KUKA KRL program: MyProgram_273().src

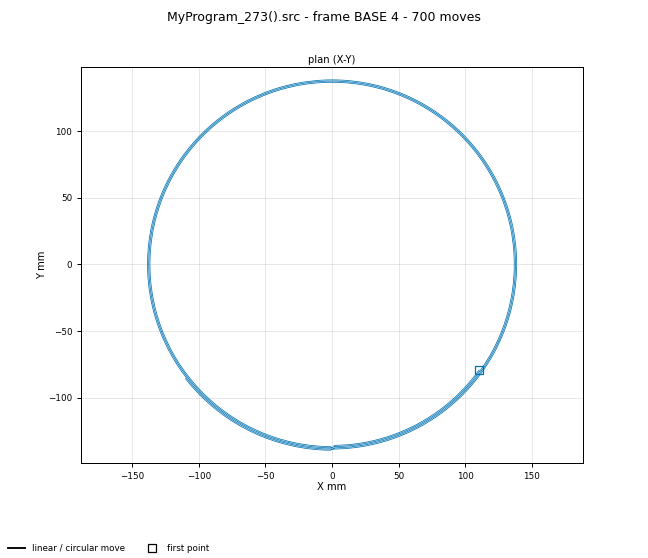
[picture p0: tool path of MyProgram_273().src in frame BASE 4, 700 of 700 moves have a stored position in this frame; points joined in program order, loops and branches not executed]
&ACCESS RVP
&REL 1
&PARAM TEMPLATE = C:\KRC\Roboter\Template\vorgabe
&PARAM EDITMASK = *
DEF MyProgram_273()
; ---- Setting reference (Base) ----
$BASE = BASE_DATA[4]

; --------------------------
; ---- Setting tool (TCP) ----
$TOOL = TOOL_DATA[3]
; --------------------------

$VEL.CP = VEL_APROX_PRINT
Startdeposition()
$VEL.CP = VEL_PRINT
LIN {X 110.2888,Y -79.2997,Z 171,A -34.2093,B 9.0943,C 0.3127,E1 9.2291,E2 485.5867} C_DIS
LIN {X 107.672,Y -82.8179,Z 171,A -36.0735,B 9.0942,C 0.3174,E1 9.226,E2 487.4547} C_DIS
LIN {X 104.9459,Y -86.2463,Z 171,A -37.9185,B 9.094,C 0.3216,E1 9.2227,E2 489.3013} C_DIS
LIN {X 101.9868,Y -89.7259,Z 171,A -39.7835,B 9.094,C 0.3246,E1 9.2193,E2 491.1605} C_DIS
LIN {X 99.052,Y -92.9557,Z 171,A -41.6097,B 9.0938,C 0.3284,E1 9.2159,E2 492.9868} C_DIS
LIN {X 95.9836,Y -96.1207,Z 171,A -43.5121,B 9.0936,C 0.3333,E1 9.2121,E2 494.8965} C_DIS
LIN {X 92.5375,Y -99.4422,Z 171,A -45.3676,B 9.0936,C 0.3339,E1 9.2084,E2 496.7335} C_DIS
LIN {X 89.5014,Y -102.1836,Z 171,A -47.1413,B 9.0934,C 0.3385,E1 9.2047,E2 498.5149} C_DIS
LIN {X 85.9377,Y -105.1981,Z 171,A -48.9197,B 9.0934,C 0.3381,E1 9.2009,E2 500.2713} C_DIS
LIN {X 82.826,Y -107.6658,Z 171,A -50.7547,B 9.0932,C 0.3448,E1 9.1968,E2 502.128} C_DIS
LIN {X 79.3157,Y -110.2774,Z 171,A -52.4701,B 9.0932,C 0.3453,E1 9.193,E2 503.8288} C_DIS
LIN {X 75.9025,Y -112.6536,Z 171,A -54.2813,B 9.093,C 0.3496,E1 9.1888,E2 505.6489} C_DIS
LIN {X 72.1992,Y -115.0623,Z 171,A -56.1436,B 9.0929,C 0.3526,E1 9.1844,E2 507.5127} C_DIS
LIN {X 69.2091,Y -116.8853,Z 171,A -57.4543,B 9.0929,C 0.3514,E1 9.1813,E2 508.8038} C_DIS
LIN {X 63.7335,Y -119.9577,Z 171,A -60.1603,B 9.0927,C 0.3567,E1 9.1747,E2 511.5193} C_DIS
LIN {X 60.3824,Y -121.6777,Z 171,A -61.7388,B 9.0927,C 0.3587,E1 9.1708,E2 513.0978} C_DIS
LIN {X 56.7536,Y -123.4119,Z 171,A -63.423,B 9.0926,C 0.3607,E1 9.1665,E2 514.7819} C_DIS
LIN {X 52.7255,Y -125.1862,Z 171,A -65.2144,B 9.0926,C 0.3617,E1 9.1619,E2 516.5666} C_DIS
LIN {X 50.0864,Y -126.2669,Z 171,A -66.5978,B 9.0923,C 0.3669,E1 9.1583,E2 517.9737} C_DIS
LIN {X 46.1854,Y -127.7433,Z 171,A -68.2377,B 9.0923,C 0.3664,E1 9.154,E2 519.6} C_DIS
LIN {X 42.2838,Y -129.0888,Z 171,A -70.0071,B 9.0923,C 0.3688,E1 9.1493,E2 521.3743} C_DIS
LIN {X 38.5569,Y -130.2496,Z 171,A -71.5883,B 9.0923,C 0.369,E1 9.1451,E2 522.9485} C_DIS
LIN {X 34.9122,Y -131.273,Z 171,A -73.1237,B 9.0923,C 0.3691,E1 9.141,E2 524.4773} C_DIS
LIN {X 31.5826,Y -132.1138,Z 171,A -74.6101,B 9.0922,C 0.3711,E1 9.137,E2 525.9694} C_DIS
LIN {X 27.5255,Y -133.0189,Z 171,A -76.3575,B 9.0922,C 0.3723,E1 9.1322,E2 527.7172} C_DIS
LIN {X 23.8817,Y -133.7204,Z 171,A -77.8272,B 9.0922,C 0.3713,E1 9.1282,E2 529.176} C_DIS
LIN {X 20.5645,Y -134.2708,Z 171,A -79.3166,B 9.0921,C 0.3736,E1 9.124,E2 530.6751} C_DIS
LIN {X 16.385,Y -134.8448,Z 171,A -81.052,B 9.0921,C 0.3736,E1 9.1193,E2 532.406} C_DIS
LIN {X 13.6701,Y -135.1485,Z 171,A -82.6176,B 9.0917,C 0.3824,E1 9.1148,E2 534.0241} C_DIS
LIN {X 9.9582,Y -135.4709,Z 171,A -83.7269,B 9.0921,C 0.3737,E1 9.1118,E2 535.0764} C_DIS
LIN {X 2.0076,Y -135.8219,Z 171,A -87.0574,B 9.0921,C 0.374,E1 9.1026,E2 538.4055} C_DIS
LIN {X 2.0076,Y -135.8219,Z 171,A -87.0574,B 9.0921,C 0.374,E1 9.1026,E2 538.4055} C_DIS
Enddeposition()
LIN {X 0.9917,Y -136.7415,Z 171,A -87.0539,B 9.0534,C 0.3716,E1 9.0639,E2 538.3927} C_DIS
Startdeposition()
$VEL.CP = VEL_PRINT
LIN {X 3.873,Y -136.6919,Z 171,A -85.7411,B 9.0534,C 0.3693,E1 9.0676,E2 537.066} C_DIS
LIN {X 6.7914,Y -136.578,Z 171,A -84.4615,B 9.0535,C 0.3678,E1 9.0711,E2 535.7785} C_DIS
LIN {X 10.0316,Y -136.3783,Z 171,A -83.129,B 9.0535,C 0.368,E1 9.0749,E2 534.4488} C_DIS
LIN {X 13.3491,Y -136.0938,Z 171,A -81.6253,B 9.0537,C 0.3652,E1 9.0791,E2 532.9305} C_DIS
LIN {X 16.9828,Y -135.6903,Z 171,A -80.2042,B 9.0536,C 0.3668,E1 9.083,E2 531.5227} C_DIS
LIN {X 20.1333,Y -135.2587,Z 171,A -78.8736,B 9.0536,C 0.3661,E1 9.0867,E2 530.1915} C_DIS
LIN {X 23.2971,Y -134.7498,Z 171,A -77.533,B 9.0536,C 0.3653,E1 9.0904,E2 528.8504} C_DIS
LIN {X 26.4717,Y -134.1623,Z 171,A -76.04,B 9.0538,C 0.3615,E1 9.0945,E2 527.3386} C_DIS
LIN {X 29.8951,Y -133.4399,Z 171,A -74.6788,B 9.0538,C 0.3626,E1 9.0982,E2 525.9898} C_DIS
LIN {X 33.2548,Y -132.6419,Z 171,A -73.4363,B 9.0536,C 0.3657,E1 9.1015,E2 524.7724} C_DIS
LIN {X 36.0325,Y -131.9164,Z 171,A -71.9412,B 9.0539,C 0.3585,E1 9.1056,E2 523.2391} C_DIS
LIN {X 39.6821,Y -130.8626,Z 171,A -70.6296,B 9.0537,C 0.3629,E1 9.109,E2 521.9621} C_DIS
LIN {X 42.4081,Y -130.007,Z 171,A -69.3026,B 9.0539,C 0.359,E1 9.1126,E2 520.6177} C_DIS
LIN {X 45.5874,Y -128.9266,Z 171,A -67.9022,B 9.0539,C 0.3576,E1 9.1163,E2 519.217} C_DIS
LIN {X 48.7566,Y -127.7617,Z 171,A -66.4946,B 9.054,C 0.3562,E1 9.12,E2 517.8093} C_DIS
LIN {X 52.3424,Y -126.3328,Z 171,A -64.8676,B 9.054,C 0.354,E1 9.1242,E2 516.1798} C_DIS
LIN {X 55.0524,Y -125.1778,Z 171,A -63.6596,B 9.0541,C 0.353,E1 9.1273,E2 514.9741} C_DIS
LIN {X 58.1724,Y -123.7588,Z 171,A -62.2327,B 9.0541,C 0.3513,E1 9.1309,E2 513.5473} C_DIS
LIN {X 61.2693,Y -122.2552,Z 171,A -60.6628,B 9.0544,C 0.3466,E1 9.1349,E2 511.9597} C_DIS
LIN {X 65.1029,Y -120.2576,Z 171,A -58.8989,B 9.0544,C 0.3449,E1 9.1392,E2 510.2003} C_DIS
LIN {X 68.8887,Y -118.1297,Z 171,A -57.0932,B 9.0545,C 0.3424,E1 9.1436,E2 508.3949} C_DIS
LIN {X 72.6202,Y -115.8731,Z 171,A -55.281,B 9.0546,C 0.3398,E1 9.1479,E2 506.583} C_DIS
LIN {X 76.291,Y -113.4899,Z 171,A -53.4633,B 9.0547,C 0.337,E1 9.1521,E2 504.7656} C_DIS
LIN {X 79.8947,Y -110.9825,Z 171,A -51.6558,B 9.0548,C 0.3344,E1 9.1562,E2 502.9605} C_DIS
LIN {X 83.4251,Y -108.3537,Z 171,A -49.8295,B 9.0549,C 0.3314,E1 9.1603,E2 501.1348} C_DIS
LIN {X 86.8762,Y -105.6068,Z 171,A -48.0005,B 9.0551,C 0.3283,E1 9.1643,E2 499.3065} C_DIS
LIN {X 90.2421,Y -102.7455,Z 171,A -46.1693,B 9.0551,C 0.3251,E1 9.1681,E2 497.476} C_DIS
LIN {X 93.5172,Y -99.7738,Z 171,A -44.3222,B 9.0553,C 0.3214,E1 9.1719,E2 495.6278} C_DIS
LIN {X 96.6961,Y -96.6961,Z 171,A -42.5051,B 9.0554,C 0.3183,E1 9.1755,E2 493.8135} C_DIS
LIN {X 99.7738,Y -93.5172,Z 171,A -40.6587,B 9.0555,C 0.3144,E1 9.1791,E2 491.9663} C_DIS
LIN {X 102.7455,Y -90.2421,Z 171,A -38.8292,B 9.0557,C 0.3108,E1 9.1825,E2 490.1379} C_DIS
LIN {X 105.6068,Y -86.8762,Z 171,A -37.0024,B 9.0557,C 0.3071,E1 9.1858,E2 488.3123} C_DIS
LIN {X 108.3537,Y -83.4251,Z 171,A -35.1793,B 9.0559,C 0.3033,E1 9.1889,E2 486.4905} C_DIS
LIN {X 110.9825,Y -79.8947,Z 171,A -33.3758,B 9.056,C 0.2998,E1 9.1919,E2 484.6903} C_DIS
LIN {X 113.4899,Y -76.291,Z 171,A -31.5625,B 9.0562,C 0.2959,E1 9.1947,E2 482.8785} C_DIS
LIN {X 115.8731,Y -72.6202,Z 171,A -29.7557,B 9.0562,C 0.2919,E1 9.1974,E2 481.0731} C_DIS
LIN {X 118.1297,Y -68.8887,Z 171,A -27.956,B 9.0564,C 0.2879,E1 9.2,E2 479.2751} C_DIS
LIN {X 120.2576,Y -65.1029,Z 171,A -26.1847,B 9.0565,C 0.2843,E1 9.2024,E2 477.508} C_DIS
LIN {X 122.2552,Y -61.2693,Z 171,A -24.4684,B 9.0566,C 0.2817,E1 9.2045,E2 475.8019} C_DIS
LIN {X 123.7588,Y -58.1724,Z 171,A -23.0371,B 9.0567,C 0.2781,E1 9.2063,E2 474.3705} C_DIS
LIN {X 125.1778,Y -55.0524,Z 171,A -21.6354,B 9.0568,C 0.275,E1 9.2079,E2 472.9717} C_DIS
LIN {X 126.6723,Y -51.5156,Z 171,A -20.0199,B 9.057,C 0.2704,E1 9.2096,E2 471.3536} C_DIS
LIN {X 127.8921,Y -48.4084,Z 171,A -18.8127,B 9.057,C 0.271,E1 9.2108,E2 470.1693} C_DIS
LIN {X 128.9266,Y -45.5874,Z 171,A -17.4388,B 9.0571,C 0.2649,E1 9.2121,E2 468.7795} C_DIS
LIN {X 130.1445,Y -41.9777,Z 171,A -15.9362,B 9.0571,C 0.2626,E1 9.2134,E2 467.287} C_DIS
LIN {X 131.0034,Y -39.2221,Z 171,A -14.6802,B 9.0573,C 0.2581,E1 9.2144,E2 466.0239} C_DIS
LIN {X 131.9164,Y -36.0325,Z 171,A -13.3137,B 9.0574,C 0.2547,E1 9.2155,E2 464.659} C_DIS
LIN {X 132.7466,Y -32.8423,Z 171,A -11.9562,B 9.0574,C 0.2514,E1 9.2164,E2 463.3031} C_DIS
LIN {X 133.4949,Y -29.6544,Z 171,A -10.4872,B 9.0577,C 0.2452,E1 9.2173,E2 461.8204} C_DIS
LIN {X 134.1623,Y -26.4717,Z 171,A -9.2693,B 9.0577,C 0.2446,E1 9.218,E2 460.6194} C_DIS
LIN {X 134.7498,Y -23.2971,Z 171,A -7.9402,B 9.0577,C 0.2413,E1 9.2186,E2 459.292} C_DIS
LIN {X 135.2587,Y -20.1333,Z 171,A -6.6214,B 9.0579,C 0.238,E1 9.2192,E2 457.9749} C_DIS
LIN {X 135.7338,Y -16.6182,Z 171,A -5.2956,B 9.0579,C 0.2374,E1 9.2197,E2 456.6678} C_DIS
LIN {X 136.0459,Y -13.8481,Z 171,A -4.0144,B 9.058,C 0.2314,E1 9.22,E2 455.3712} C_DIS
LIN {X 136.3272,Y -10.7317,Z 171,A -2.6901,B 9.0581,C 0.2273,E1 9.2204,E2 454.044} C_DIS
LIN {X 136.5356,Y -7.6359,Z 171,A -1.4498,B 9.0581,C 0.2249,E1 9.2206,E2 452.81} C_DIS
LIN {X 136.6728,Y -4.5627,Z 171,A -0.0223,B 9.0584,C 0.2179,E1 9.2207,E2 451.3637} C_DIS
LIN {X 136.7472,Y -0.5669,Z 171,A 1.3911,B 9.0584,C 0.2191,E1 9.2207,E2 449.9817} C_DIS
LIN {X 136.7291,Y 2.201,Z 171,A 2.6312,B 9.0584,C 0.2138,E1 9.2207,E2 448.7303} C_DIS
LIN {X 136.6458,Y 5.2551,Z 171,A 3.866,B 9.0585,C 0.2112,E1 9.2207,E2 447.5} C_DIS
LIN {X 136.4833,Y 8.4834,Z 171,A 5.2015,B 9.0585,C 0.2077,E1 9.2204,E2 446.1657} C_DIS
LIN {X 136.239,Y 11.7759,Z 171,A 6.6115,B 9.0587,C 0.2031,E1 9.2201,E2 444.7511} C_DIS
LIN {X 135.8775,Y 15.4133,Z 171,A 8.0744,B 9.0587,C 0.2002,E1 9.2196,E2 443.2956} C_DIS
LIN {X 135.4537,Y 18.7684,Z 171,A 9.3927,B 9.0588,C 0.1984,E1 9.2192,E2 441.9885} C_DIS
LIN {X 135.014,Y 21.7137,Z 171,A 10.832,B 9.059,C 0.1905,E1 9.2185,E2 440.524} C_DIS
LIN {X 134.3733,Y 25.3678,Z 171,A 12.2748,B 9.059,C 0.1886,E1 9.2178,E2 439.0939} C_DIS
LIN {X 133.4949,Y 29.6544,Z 171,A 14.0413,B 9.059,C 0.1849,E1 9.2168,E2 437.3344} C_DIS
LIN {X 132.6344,Y 33.2844,Z 171,A 15.5539,B 9.0591,C 0.1817,E1 9.2158,E2 435.8268} C_DIS
LIN {X 131.8569,Y 36.2452,Z 171,A 16.8542,B 9.0592,C 0.1777,E1 9.2149,E2 434.5233} C_DIS
LIN {X 131.0034,Y 39.2221,Z 171,A 18.1264,B 9.0592,C 0.1747,E1 9.2139,E2 433.2533} C_DIS
LIN {X 129.8916,Y 42.7547,Z 171,A 19.6534,B 9.0594,C 0.171,E1 9.2126,E2 431.7282} C_DIS
LIN {X 128.9266,Y 45.5874,Z 171,A 20.8926,B 9.0594,C 0.1679,E1 9.2114,E2 430.49} C_DIS
LIN {X 127.7617,Y 48.7566,Z 171,A 22.375,B 9.0595,C 0.1626,E1 9.2099,E2 428.9981} C_DIS
LIN {X 126.5122,Y 51.9128,Z 171,A 23.6906,B 9.0595,C 0.1612,E1 9.2086,E2 427.6949} C_DIS
LIN {X 124.9735,Y 55.5093,Z 171,A 25.2436,B 9.0595,C 0.1588,E1 9.2069,E2 426.1515} C_DIS
LIN {X 123.5373,Y 58.636,Z 171,A 26.5408,B 9.0595,C 0.1582,E1 9.2054,E2 424.8714} C_DIS
LIN {X 122.0945,Y 61.5849,Z 171,A 28.0933,B 9.0597,C 0.1507,E1 9.2034,E2 423.2959} C_DIS
LIN {X 120.276,Y 65.0685,Z 171,A 29.8184,B 9.0598,C 0.1448,E1 9.2011,E2 421.5601} C_DIS
LIN {X 118.0845,Y 68.9655,Z 171,A 31.6414,B 9.0598,C 0.1412,E1 9.1986,E2 419.7423} C_DIS
LIN {X 115.8731,Y 72.6202,Z 171,A 33.4486,B 9.0599,C 0.1365,E1 9.1959,E2 417.932} C_DIS
LIN {X 113.4899,Y 76.291,Z 171,A 35.2409,B 9.0599,C 0.133,E1 9.1932,E2 416.1439} C_DIS
LIN {X 110.9825,Y 79.8947,Z 171,A 37.0651,B 9.06,C 0.129,E1 9.1902,E2 414.3206} C_DIS
LIN {X 108.3537,Y 83.4251,Z 171,A 38.8844,B 9.06,C 0.1254,E1 9.1872,E2 412.5036} C_DIS
LIN {X 105.6068,Y 86.8762,Z 171,A 40.6901,B 9.0601,C 0.1222,E1 9.184,E2 410.7024} C_DIS
LIN {X 102.7455,Y 90.2421,Z 171,A 42.5256,B 9.0601,C 0.1185,E1 9.1807,E2 408.8681} C_DIS
LIN {X 99.7738,Y 93.5172,Z 171,A 44.3659,B 9.0602,C 0.1149,E1 9.1772,E2 407.0287} C_DIS
LIN {X 96.6961,Y 96.6961,Z 171,A 46.1837,B 9.0602,C 0.1119,E1 9.1736,E2 405.2147} C_DIS
LIN {X 93.5172,Y 99.7738,Z 171,A 48.0321,B 9.0603,C 0.1083,E1 9.1699,E2 403.3664} C_DIS
LIN {X 90.2421,Y 102.7455,Z 171,A 49.8651,B 9.0603,C 0.1052,E1 9.1661,E2 401.5354} C_DIS
LIN {X 86.8172,Y 105.655,Z 171,A 51.7094,B 9.0603,C 0.1026,E1 9.1621,E2 399.6955} C_DIS
LIN {X 83.4182,Y 108.3589,Z 171,A 53.527,B 9.0604,C 0.0995,E1 9.1581,E2 397.8777} C_DIS
LIN {X 79.8947,Y 110.9825,Z 171,A 55.3362,B 9.0604,C 0.097,E1 9.154,E2 396.0721} C_DIS
LIN {X 76.291,Y 113.4899,Z 171,A 57.158,B 9.0604,C 0.0944,E1 9.1499,E2 394.2522} C_DIS
LIN {X 72.6202,Y 115.8731,Z 171,A 58.9746,B 9.0604,C 0.092,E1 9.1456,E2 392.4375} C_DIS
LIN {X 68.8887,Y 118.1297,Z 171,A 60.7852,B 9.0605,C 0.0897,E1 9.1412,E2 390.6289} C_DIS
LIN {X 65.1029,Y 120.2576,Z 171,A 62.5684,B 9.0605,C 0.0879,E1 9.1369,E2 388.85} C_DIS
LIN {X 61.2693,Y 122.2552,Z 171,A 64.2972,B 9.0605,C 0.0873,E1 9.1326,E2 387.1314} C_DIS
LIN {X 57.8326,Y 123.9159,Z 171,A 65.9138,B 9.0605,C 0.085,E1 9.1285,E2 385.5126} C_DIS
LIN {X 54.7106,Y 125.3257,Z 171,A 67.1708,B 9.0605,C 0.087,E1 9.1254,E2 384.2777} C_DIS
LIN {X 51.9128,Y 126.5122,Z 171,A 68.5727,B 9.0605,C 0.083,E1 9.1217,E2 382.8601} C_DIS
LIN {X 48.7566,Y 127.7617,Z 171,A 69.9852,B 9.0605,C 0.0817,E1 9.118,E2 381.4489} C_DIS
LIN {X 45.1805,Y 129.0676,Z 171,A 71.5897,B 9.0606,C 0.08,E1 9.1138,E2 379.8434} C_DIS
LIN {X 41.8719,Y 130.1783,Z 171,A 72.9371,B 9.0606,C 0.0811,E1 9.1103,E2 378.5103} C_DIS
LIN {X 39.2221,Y 131.0034,Z 171,A 74.179,B 9.0606,C 0.0785,E1 9.1069,E2 377.2589} C_DIS
LIN {X 36.0325,Y 131.9164,Z 171,A 75.7095,B 9.0606,C 0.0746,E1 9.1028,E2 375.7114} C_DIS
LIN {X 32.348,Y 132.8657,Z 171,A 76.9585,B 9.0606,C 0.0805,E1 9.0995,E2 374.5051} C_DIS
LIN {X 29.6544,Y 133.4949,Z 171,A 78.3001,B 9.0606,C 0.0761,E1 9.0958,E2 373.1414} C_DIS
LIN {X 26.4717,Y 134.1623,Z 171,A 79.8045,B 9.0606,C 0.0725,E1 9.0916,E2 371.62} C_DIS
LIN {X 22.7916,Y 134.8341,Z 171,A 81.2261,B 9.0606,C 0.0746,E1 9.0878,E2 370.2167} C_DIS
LIN {X 18.5562,Y 135.4841,Z 171,A 83.1326,B 9.0606,C 0.0717,E1 9.0825,E2 368.2971} C_DIS
LIN {X 15.4133,Y 135.8775,Z 171,A 84.3274,B 9.0606,C 0.0739,E1 9.0792,E2 367.1191} C_DIS
LIN {X 12.2875,Y 136.1958,Z 171,A 85.8008,B 9.0606,C 0.0705,E1 9.0751,E2 365.6269} C_DIS
LIN {X 8.373,Y 136.4902,Z 171,A 87.2861,B 9.0606,C 0.0734,E1 9.071,E2 364.1617} C_DIS
LIN {X 5.2551,Y 136.6458,Z 171,A 88.5562,B 9.0606,C 0.074,E1 9.0674,E2 362.8968} C_DIS
LIN {X 2.201,Y 136.7291,Z 171,A 89.8336,B 9.0606,C 0.074,E1 9.0639,E2 361.6203} C_DIS
LIN {X -0.8306,Y 136.7443,Z 171,A 91.1056,B 9.0606,C 0.074,E1 9.0603,E2 360.3487} C_DIS
LIN {X -3.9636,Y 136.6894,Z 171,A 92.5121,B 9.0606,C 0.0723,E1 9.0564,E2 358.9313} C_DIS
LIN {X -7.6359,Y 136.5356,Z 171,A 93.9932,B 9.0606,C 0.0737,E1 9.0523,E2 357.4583} C_DIS
LIN {X -10.7317,Y 136.3272,Z 171,A 95.2974,B 9.0606,C 0.0739,E1 9.0486,E2 356.1543} C_DIS
LIN {X -13.8481,Y 136.0459,Z 171,A 96.6132,B 9.0606,C 0.0742,E1 9.045,E2 354.8386} C_DIS
LIN {X -16.9828,Y 135.6903,Z 171,A 98.0979,B 9.0606,C 0.0716,E1 9.0408,E2 353.3347} C_DIS
LIN {X -21.7137,Y 135.014,Z 171,A 99.951,B 9.0606,C 0.0753,E1 9.0357,E2 351.5011} C_DIS
LIN {X -24.8832,Y 134.4659,Z 171,A 101.3051,B 9.0606,C 0.0759,E1 9.032,E2 350.147} C_DIS
LIN {X -28.0622,Y 133.8386,Z 171,A 102.6696,B 9.0606,C 0.0766,E1 9.0283,E2 348.7826} C_DIS
LIN {X -31.5432,Y 133.0597,Z 171,A 104.1553,B 9.0606,C 0.0778,E1 9.0242,E2 347.2988} C_DIS
LIN {X -34.4373,Y 132.3418,Z 171,A 105.4285,B 9.0606,C 0.0783,E1 9.0208,E2 346.0235} C_DIS
LIN {X -37.6276,Y 131.4703,Z 171,A 106.9347,B 9.0606,C 0.0772,E1 9.0167,E2 344.5035} C_DIS
LIN {X -41.3181,Y 130.3552,Z 171,A 108.463,B 9.0606,C 0.0802,E1 9.0127,E2 342.987} C_DIS
LIN {X -43.9988,Y 129.4773,Z 171,A 109.6382,B 9.0606,C 0.0814,E1 9.0096,E2 341.8136} C_DIS
LIN {X -47.1734,Y 128.3547,Z 171,A 111.0588,B 9.0606,C 0.0827,E1 9.0058,E2 340.3929} C_DIS
LIN {X -50.3366,Y 127.1475,Z 171,A 112.4877,B 9.0606,C 0.084,E1 9.0021,E2 338.9637} C_DIS
LIN {X -53.4849,Y 125.8556,Z 171,A 114.0521,B 9.0606,C 0.0831,E1 8.998,E2 337.3835} C_DIS
LIN {X -56.8116,Y 124.388,Z 171,A 115.3785,B 9.0606,C 0.0885,E1 8.9947,E2 336.0824} C_DIS
LIN {X -59.7239,Y 123.0175,Z 171,A 116.8198,B 9.0606,C 0.0886,E1 8.9911,E2 334.6309} C_DIS
LIN {X -62.808,Y 121.4719,Z 171,A 118.4237,B 9.0606,C 0.0877,E1 8.987,E2 333.0087} C_DIS
LIN {X -66.6233,Y 119.422,Z 171,A 120.1989,B 9.0606,C 0.091,E1 8.9827,E2 331.2399} C_DIS
LIN {X -70.3881,Y 117.2424,Z 171,A 122.039,B 9.0605,C 0.0934,E1 8.9783,E2 329.3992} C_DIS
LIN {X -74.0961,Y 114.9349,Z 171,A 123.8868,B 9.0605,C 0.096,E1 8.9739,E2 327.5508} C_DIS
LIN {X -77.7408,Y 112.5017,Z 171,A 125.7571,B 9.0605,C 0.0984,E1 8.9696,E2 325.6779} C_DIS
LIN {X -81.316,Y 109.9453,Z 171,A 127.6025,B 9.0604,C 0.1015,E1 8.9654,E2 323.8338} C_DIS
LIN {X -84.8154,Y 107.2689,Z 171,A 129.4839,B 9.0604,C 0.1043,E1 8.9613,E2 321.9497} C_DIS
LIN {X -88.2727,Y 104.4421,Z 171,A 131.3628,B 9.0604,C 0.1077,E1 8.9572,E2 320.0716} C_DIS
LIN {X -91.5633,Y 101.5698,Z 171,A 133.2115,B 9.0603,C 0.1109,E1 8.9534,E2 318.2225} C_DIS
LIN {X -94.8006,Y 98.5552,Z 171,A 135.0865,B 9.0603,C 0.1143,E1 8.9496,E2 316.3466} C_DIS
LIN {X -97.9396,Y 95.4364,Z 171,A 136.9783,B 9.0602,C 0.1175,E1 8.9459,E2 314.452} C_DIS
LIN {X -100.9754,Y 92.2184,Z 171,A 138.8389,B 9.0602,C 0.1214,E1 8.9423,E2 312.5924} C_DIS
LIN {X -103.9035,Y 88.9063,Z 171,A 140.7299,B 9.0602,C 0.1248,E1 8.9389,E2 310.6985} C_DIS
LIN {X -106.7548,Y 85.4613,Z 171,A 142.613,B 9.06,C 0.1289,E1 8.9355,E2 308.8161} C_DIS
LIN {X -109.4196,Y 82.0221,Z 171,A 144.4705,B 9.06,C 0.1326,E1 8.9324,E2 306.9561} C_DIS
LIN {X -112.0002,Y 78.4616,Z 171,A 146.3403,B 9.06,C 0.1365,E1 8.9294,E2 305.0848} C_DIS
LIN {X -114.4775,Y 74.8007,Z 171,A 148.1925,B 9.0599,C 0.1411,E1 8.9265,E2 303.2346} C_DIS
LIN {X -116.791,Y 71.1345,Z 171,A 150.0578,B 9.0599,C 0.1448,E1 8.9238,E2 301.3651} C_DIS
LIN {X -118.9964,Y 67.3805,Z 171,A 151.9067,B 9.0597,C 0.149,E1 8.9212,E2 299.515} C_DIS
LIN {X -120.6909,Y 64.2953,Z 171,A 153.4263,B 9.0597,C 0.152,E1 8.9192,E2 297.9915} C_DIS
LIN {X -122.2552,Y 61.2693,Z 171,A 154.7436,B 9.0596,C 0.1576,E1 8.9175,E2 296.6892} C_DIS
LIN {X -123.7588,Y 58.1724,Z 171,A 156.2065,B 9.0596,C 0.1611,E1 8.9158,E2 295.2253} C_DIS
LIN {X -125.1778,Y 55.0524,Z 171,A 157.6631,B 9.0595,C 0.1646,E1 8.9141,E2 293.7676} C_DIS
LIN {X -126.6252,Y 51.6322,Z 171,A 159.127,B 9.0594,C 0.1703,E1 8.9125,E2 292.3167} C_DIS
LIN {X -127.7617,Y 48.7566,Z 171,A 160.556,B 9.0594,C 0.1716,E1 8.9111,E2 290.8726} C_DIS
LIN {X -128.9266,Y 45.5874,Z 171,A 161.9912,B 9.0593,C 0.1752,E1 8.9097,E2 289.4364} C_DIS
LIN {X -130.007,Y 42.4081,Z 171,A 163.5064,B 9.0593,C 0.1773,E1 8.9084,E2 287.9092} C_DIS
LIN {X -131.0034,Y 39.2221,Z 171,A 164.8381,B 9.0591,C 0.1823,E1 8.9073,E2 286.5873} C_DIS
LIN {X -131.9164,Y 36.0325,Z 171,A 166.2486,B 9.0591,C 0.1858,E1 8.9062,E2 285.1756} C_DIS
LIN {X -132.7466,Y 32.8423,Z 171,A 167.6503,B 9.059,C 0.1894,E1 8.9053,E2 283.7728} C_DIS
LIN {X -133.5384,Y 29.453,Z 171,A 169.052,B 9.0589,C 0.1945,E1 8.9044,E2 282.3795} C_DIS
LIN {X -134.1623,Y 26.4717,Z 171,A 170.4252,B 9.0589,C 0.1965,E1 8.9036,E2 280.9957} C_DIS
LIN {X -134.7498,Y 23.2971,Z 171,A 171.798,B 9.0588,C 0.2001,E1 8.903,E2 279.6217} C_DIS
LIN {X -135.2587,Y 20.1333,Z 171,A 173.2816,B 9.0588,C 0.2016,E1 8.9023,E2 278.122} C_DIS
LIN {X -135.7345,Y 16.6117,Z 171,A 174.664,B 9.0586,C 0.2077,E1 8.9018,E2 276.7542} C_DIS
LIN {X -136.0459,Y 13.8481,Z 171,A 175.854,B 9.0586,C 0.2106,E1 8.9015,E2 275.5624} C_DIS
LIN {X -136.3272,Y 10.7317,Z 171,A 177.1845,B 9.0584,C 0.2141,E1 8.9012,E2 274.2307} C_DIS
LIN {X -136.5356,Y 7.6359,Z 171,A 178.6029,B 9.0584,C 0.2159,E1 8.9009,E2 272.7989} C_DIS
LIN {X -136.6919,Y 3.873,Z 171,A -179.8678,B 9.0583,C 0.2213,E1 8.9008,E2 271.277} C_DIS
LIN {X -136.751,Y 0,Z 171,A -178.0171,B 9.0583,C 0.2223,E1 8.9008,E2 269.3996} C_DIS
LIN {X -136.6919,Y -3.873,Z 171,A -176.6214,B 9.058,C 0.2307,E1 8.9008,E2 268.0336} C_DIS
LIN {X -136.578,Y -6.7914,Z 171,A -175.3065,B 9.058,C 0.2328,E1 8.901,E2 266.7085} C_DIS
LIN {X -136.3509,Y -10.4062,Z 171,A -173.6956,B 9.058,C 0.2356,E1 8.9013,E2 265.0873} C_DIS
LIN {X -136.0459,Y -13.8481,Z 171,A -172.3268,B 9.0578,C 0.2411,E1 8.9017,E2 263.7296} C_DIS
LIN {X -135.6397,Y -17.3688,Z 171,A -170.7725,B 9.0577,C 0.2442,E1 8.9022,E2 262.168} C_DIS
LIN {X -135.1759,Y -20.6683,Z 171,A -169.3638,B 9.0576,C 0.248,E1 8.9028,E2 260.7588} C_DIS
LIN {X -134.4659,Y -24.8832,Z 171,A -167.5701,B 9.0575,C 0.253,E1 8.9037,E2 258.9664} C_DIS
LIN {X -133.7222,Y -28.6015,Z 171,A -165.993,B 9.0573,C 0.2577,E1 8.9046,E2 257.392} C_DIS
LIN {X -133.0445,Y -31.6062,Z 171,A -164.7795,B 9.0572,C 0.2626,E1 8.9053,E2 256.1892} C_DIS
LIN {X -132.3418,Y -34.4373,Z 171,A -163.396,B 9.0572,C 0.2634,E1 8.9063,E2 254.7865} C_DIS
LIN {X -131.4703,Y -37.6276,Z 171,A -161.9862,B 9.0571,C 0.2668,E1 8.9073,E2 253.3748} C_DIS
LIN {X -130.5157,Y -40.8158,Z 171,A -160.5124,B 9.057,C 0.2693,E1 8.9085,E2 251.8922} C_DIS
LIN {X -129.4773,Y -43.9988,Z 171,A -159.141,B 9.0569,C 0.2737,E1 8.9098,E2 250.5257} C_DIS
LIN {X -128.3547,Y -47.1734,Z 171,A -157.6095,B 9.0569,C 0.2754,E1 8.9112,E2 248.9801} C_DIS
LIN {X -127.1475,Y -50.3366,Z 171,A -156.1155,B 9.0567,C 0.2779,E1 8.9128,E2 247.4776} C_DIS
LIN {X -125.6229,Y -54.023,Z 171,A -154.5674,B 9.0565,C 0.2844,E1 8.9144,E2 245.946} C_DIS
LIN {X -124.4789,Y -56.6151,Z 171,A -153.3598,B 9.0565,C 0.2872,E1 8.9158,E2 244.7368} C_DIS
LIN {X -122.8306,Y -60.1029,Z 171,A -151.6968,B 9.0563,C 0.2905,E1 8.9178,E2 243.0689} C_DIS
LIN {X -121.4719,Y -62.808,Z 171,A -150.3396,B 9.0563,C 0.2923,E1 8.9196,E2 241.7014} C_DIS
LIN {X -119.422,Y -66.6233,Z 171,A -148.497,B 9.0561,C 0.2963,E1 8.922,E2 239.8563} C_DIS
LIN {X -117.2424,Y -70.3881,Z 171,A -146.6469,B 9.0561,C 0.3003,E1 8.9247,E2 238.0038} C_DIS
LIN {X -114.9349,Y -74.0961,Z 171,A -144.7904,B 9.0559,C 0.3042,E1 8.9275,E2 236.145} C_DIS
LIN {X -112.5017,Y -77.7408,Z 171,A -142.9071,B 9.0558,C 0.3077,E1 8.9304,E2 234.2566} C_DIS
LIN {X -109.9453,Y -81.316,Z 171,A -141.0616,B 9.0556,C 0.3119,E1 8.9335,E2 232.4115} C_DIS
LIN {X -107.2689,Y -84.8154,Z 171,A -139.1758,B 9.0556,C 0.3153,E1 8.9367,E2 230.5215} C_DIS
LIN {X -104.4235,Y -88.2946,Z 171,A -137.2888,B 9.0554,C 0.3193,E1 8.9401,E2 228.6348} C_DIS
LIN {X -101.5698,Y -91.5633,Z 171,A -135.4437,B 9.0553,C 0.3226,E1 8.9435,E2 226.787} C_DIS
LIN {X -98.5552,Y -94.8006,Z 171,A -133.5686,B 9.0551,C 0.326,E1 8.9471,E2 224.9099} C_DIS
LIN {X -95.4364,Y -97.9396,Z 171,A -131.6724,B 9.0551,C 0.3289,E1 8.9509,E2 223.009} C_DIS
LIN {X -92.2184,Y -100.9754,Z 171,A -129.8205,B 9.0549,C 0.3324,E1 8.9547,E2 221.1577} C_DIS
LIN {X -88.9052,Y -103.9044,Z 171,A -127.9336,B 9.0549,C 0.3352,E1 8.9587,E2 219.267} C_DIS
LIN {X -85.4906,Y -106.7315,Z 171,A -126.0491,B 9.0547,C 0.338,E1 8.9627,E2 217.3795} C_DIS
LIN {X -82.0221,Y -109.4196,Z 171,A -124.2182,B 9.0546,C 0.3412,E1 8.9668,E2 215.55} C_DIS
LIN {X -78.4616,Y -112.0002,Z 171,A -122.3448,B 9.0545,C 0.3435,E1 8.9711,E2 213.6729} C_DIS
LIN {X -74.8303,Y -114.4582,Z 171,A -120.5084,B 9.0544,C 0.3463,E1 8.9753,E2 211.8369} C_DIS
LIN {X -71.0992,Y -116.8124,Z 171,A -118.6414,B 9.0544,C 0.3486,E1 8.9798,E2 209.9678} C_DIS
LIN {X -67.3463,Y -119.0156,Z 171,A -116.8055,B 9.0542,C 0.3508,E1 8.9842,E2 208.1303} C_DIS
LIN {X -64.3398,Y -120.6676,Z 171,A -115.4538,B 9.0541,C 0.3543,E1 8.9875,E2 206.7896} C_DIS
LIN {X -61.1881,Y -122.2953,Z 171,A -113.9926,B 9.054,C 0.3565,E1 8.9912,E2 205.3316} C_DIS
LIN {X -57.7374,Y -123.9599,Z 171,A -112.4088,B 9.054,C 0.3588,E1 8.9951,E2 203.7505} C_DIS
LIN {X -55.0524,Y -125.1778,Z 171,A -111.1031,B 9.054,C 0.3588,E1 8.9985,E2 202.4357} C_DIS
LIN {X -51.9128,Y -126.5122,Z 171,A -109.6671,B 9.0539,C 0.3601,E1 9.0022,E2 200.9988} C_DIS
LIN {X -48.7566,Y -127.7617,Z 171,A -108.1652,B 9.0539,C 0.3599,E1 9.0061,E2 199.4866} C_DIS
LIN {X -45.3402,Y -129.0123,Z 171,A -106.6636,B 9.0538,C 0.3617,E1 9.0101,E2 197.9877} C_DIS
LIN {X -42.4081,Y -130.007,Z 171,A -105.4073,B 9.0538,C 0.3635,E1 9.0134,E2 196.7365} C_DIS
LIN {X -39.2221,Y -131.0034,Z 171,A -103.8629,B 9.0538,C 0.3617,E1 9.0176,E2 195.1732} C_DIS
LIN {X -35.9229,Y -131.9456,Z 171,A -102.606,B 9.0536,C 0.3661,E1 9.0209,E2 193.939} C_DIS
LIN {X -32.8423,Y -132.7466,Z 171,A -101.2275,B 9.0536,C 0.3661,E1 9.0246,E2 192.5545} C_DIS
LIN {X -29.6544,Y -133.4949,Z 171,A -99.7655,B 9.0536,C 0.365,E1 9.0287,E2 191.0807} C_DIS
LIN {X -25.9986,Y -134.2527,Z 171,A -98.2843,B 9.0536,C 0.3674,E1 9.0327,E2 189.6096} C_DIS
LIN {X -23.2971,Y -134.7498,Z 171,A -97.1361,B 9.0536,C 0.3679,E1 9.0358,E2 188.4615} C_DIS
LIN {X -19.5637,Y -135.3401,Z 171,A -95.7663,B 9.0534,C 0.3726,E1 9.0396,E2 187.1184} C_DIS
LIN {X -16.9828,Y -135.6903,Z 171,A -94.4614,B 9.0535,C 0.3686,E1 9.0432,E2 185.786} C_DIS
LIN {X -13.8481,Y -136.0459,Z 171,A -93.1406,B 9.0535,C 0.3689,E1 9.0469,E2 184.4648} C_DIS
LIN {X -10.7317,Y -136.3272,Z 171,A -91.831,B 9.0535,C 0.3691,E1 9.0506,E2 183.1548} C_DIS
LIN {X -7.6359,Y -136.5356,Z 171,A -90.5328,B 9.0535,C 0.3692,E1 9.0542,E2 181.8563} C_DIS
LIN {X -4.5627,Y -136.6728,Z 171,A -89.2468,B 9.0535,C 0.3692,E1 9.0578,E2 180.5702} C_DIS
LIN {X -1.5143,Y -136.7405,Z 171,A -87.8177,B 9.0536,C 0.3661,E1 9.0618,E2 179.121} C_DIS
LIN {X -1.5143,Y -136.7405,Z 171,A -87.8177,B 9.0536,C 0.3661,E1 9.0618,E2 179.121} C_DIS
Enddeposition()
LIN {X 0.999,Y -137.6517,Z 171,A -87.1205,B 9.0143,C 0.3793,E1 9.0247,E2 178.514} C_DIS
Startdeposition()
$VEL.CP = VEL_PRINT
LIN {X -2.0065,Y -137.6428,Z 171,A -88.768,B 9.0139,C 0.3874,E1 9.02,E2 180.2128} C_DIS
LIN {X -5.8902,Y -137.532,Z 171,A -90.468,B 9.0139,C 0.3891,E1 9.0152,E2 181.9242} C_DIS
LIN {X -10.1042,Y -137.2857,Z 171,A -92.1089,B 9.0139,C 0.3867,E1 9.0107,E2 183.5509} C_DIS
LIN {X -14.2208,Y -136.9214,Z 171,A -94.4711,B 9.0134,C 0.399,E1 9.0039,E2 185.9952} C_DIS
LIN {X -19.3526,Y -136.2898,Z 171,A -95.7056,B 9.0142,C 0.3805,E1 9.0008,E2 187.114} C_DIS
LIN {X -25.3246,Y -135.3084,Z 171,A -98.3818,B 9.0142,C 0.3827,E1 8.9934,E2 189.8112} C_DIS
LIN {X -29.2332,Y -134.5171,Z 171,A -100.2355,B 9.014,C 0.3857,E1 8.9882,E2 191.6901} C_DIS
LIN {X -35.4266,Y -133.0201,Z 171,A -102.5256,B 9.0144,C 0.3772,E1 8.9821,E2 193.9347} C_DIS
LIN {X -38.8817,Y -132.0516,Z 171,A -104.3105,B 9.0142,C 0.3818,E1 8.9772,E2 195.757} C_DIS
LIN {X -42.1299,Y -131.0515,Z 171,A -105.7438,B 9.0142,C 0.381,E1 8.9734,E2 197.193} C_DIS
LIN {X -45.8425,Y -129.8016,Z 171,A -107.5224,B 9.0142,C 0.3825,E1 8.9687,E2 198.9907} C_DIS
LIN {X -49.6466,Y -128.3924,Z 171,A -109.1583,B 9.0142,C 0.3799,E1 8.9644,E2 200.6201} C_DIS
LIN {X -53.1216,Y -126.9939,Z 171,A -110.7295,B 9.0142,C 0.3786,E1 8.9603,E2 202.1929} C_DIS
LIN {X -57.3013,Y -125.1645,Z 171,A -112.6269,B 9.0144,C 0.3766,E1 8.9555,E2 204.0901} C_DIS
LIN {X -60.7318,Y -123.5354,Z 171,A -114.1955,B 9.0144,C 0.3745,E1 8.9516,E2 205.6572} C_DIS
LIN {X -63.9609,Y -121.8947,Z 171,A -115.9377,B 9.0144,C 0.377,E1 8.9472,E2 207.4291} C_DIS
LIN {X -66.8955,Y -120.3118,Z 171,A -117.0895,B 9.0146,C 0.3708,E1 8.9444,E2 208.5511} C_DIS
LIN {X -70.4874,Y -118.243,Z 171,A -118.8986,B 9.0146,C 0.37,E1 8.94,E2 210.3707} C_DIS
LIN {X -74.4691,Y -115.777,Z 171,A -120.8289,B 9.0148,C 0.3669,E1 8.9355,E2 212.2984} C_DIS
LIN {X -78.1503,Y -113.3247,Z 171,A -122.7382,B 9.0148,C 0.3653,E1 8.931,E2 214.216} C_DIS
LIN {X -81.8747,Y -110.6643,Z 171,A -124.7453,B 9.0148,C 0.364,E1 8.9265,E2 216.2357} C_DIS
LIN {X -85.817,Y -107.6351,Z 171,A -126.7236,B 9.0151,C 0.3589,E1 8.9222,E2 218.2021} C_DIS
LIN {X -89.312,Y -104.7534,Z 171,A -128.6378,B 9.0152,C 0.356,E1 8.9181,E2 220.1195} C_DIS
LIN {X -92.753,Y -101.7195,Z 171,A -130.5296,B 9.0154,C 0.3522,E1 8.9141,E2 222.0085} C_DIS
LIN {X -95.9623,Y -98.6975,Z 171,A -132.4485,B 9.0154,C 0.3501,E1 8.9102,E2 223.9375} C_DIS
LIN {X -98.5779,Y -96.0856,Z 171,A -134.025,B 9.0155,C 0.3477,E1 8.9071,E2 225.5182} C_DIS
LIN {X -101.6495,Y -92.8301,Z 171,A -135.9417,B 9.0156,C 0.3448,E1 8.9035,E2 227.441} C_DIS
LIN {X -104.2352,Y -89.9161,Z 171,A -137.4907,B 9.0158,C 0.3402,E1 8.9007,E2 228.9803} C_DIS
LIN {X -107.0382,Y -86.5605,Z 171,A -139.3421,B 9.0159,C 0.3367,E1 8.8974,E2 230.8348} C_DIS
LIN {X -109.6717,Y -83.1991,Z 171,A -141.1727,B 9.0161,C 0.3337,E1 8.8942,E2 232.6713} C_DIS
LIN {X -112.3208,Y -79.5864,Z 171,A -143.0719,B 9.0161,C 0.33,E1 8.8911,E2 234.5739} C_DIS
LIN {X -114.9855,Y -75.6849,Z 171,A -145.0314,B 9.0164,C 0.3253,E1 8.8881,E2 236.5315} C_DIS
LIN {X -117.4922,Y -71.7324,Z 171,A -147.0075,B 9.0165,C 0.321,E1 8.8852,E2 238.5101} C_DIS
LIN {X -119.7219,Y -67.9459,Z 171,A -148.7613,B 9.0167,C 0.3153,E1 8.8827,E2 240.2534} C_DIS
LIN {X -122.1817,Y -63.4144,Z 171,A -150.9257,B 9.0169,C 0.3102,E1 8.8799,E2 242.4189} C_DIS
LIN {X -123.5581,Y -60.6859,Z 171,A -152.2181,B 9.0169,C 0.3073,E1 8.8783,E2 243.7129} C_DIS
LIN {X -124.9425,Y -57.7815,Z 171,A -153.6327,B 9.0171,C 0.3051,E1 8.8766,E2 245.1361} C_DIS
LIN {X -126.4786,Y -54.3379,Z 171,A -155.1801,B 9.0172,C 0.3006,E1 8.8748,E2 246.6797} C_DIS
LIN {X -127.756,Y -51.262,Z 171,A -156.6168,B 9.0173,C 0.2978,E1 8.8733,E2 248.1217} C_DIS
LIN {X -129.1906,Y -47.5372,Z 171,A -158.3747,B 9.0173,C 0.2949,E1 8.8716,E2 249.8906} C_DIS
LIN {X -130.6906,Y -43.2364,Z 171,A -160.2028,B 9.0176,C 0.2886,E1 8.8699,E2 251.7088} C_DIS
LIN {X -131.7682,Y -39.8336,Z 171,A -161.7374,B 9.0176,C 0.2854,E1 8.8687,E2 253.2484} C_DIS
LIN {X -132.8595,Y -36.0288,Z 171,A -163.4527,B 9.0178,C 0.2819,E1 8.8674,E2 254.9709} C_DIS
LIN {X -133.8205,Y -32.2716,Z 171,A -165.0378,B 9.018,C 0.2769,E1 8.8663,E2 256.551} C_DIS
LIN {X -134.6073,Y -28.8155,Z 171,A -166.5183,B 9.018,C 0.2729,E1 8.8654,E2 258.0309} C_DIS
LIN {X -135.3025,Y -25.3553,Z 171,A -168.1539,B 9.0181,C 0.2715,E1 8.8645,E2 259.6861} C_DIS
LIN {X -136.0197,Y -21.168,Z 171,A -169.8257,B 9.0183,C 0.2648,E1 8.8638,E2 261.3444} C_DIS
LIN {X -136.5146,Y -17.698,Z 171,A -171.3127,B 9.0184,C 0.2611,E1 8.8632,E2 262.8336} C_DIS
LIN {X -136.9376,Y -14.0705,Z 171,A -172.9281,B 9.0185,C 0.2583,E1 8.8627,E2 264.4595} C_DIS
LIN {X -137.2811,Y -10.1676,Z 171,A -174.5261,B 9.0187,C 0.2531,E1 8.8624,E2 266.052} C_DIS
LIN {X -137.499,Y -6.6028,Z 171,A -175.9964,B 9.0187,C 0.2485,E1 8.8621,E2 267.5189} C_DIS
LIN {X -137.6202,Y -3.2403,Z 171,A -177.5494,B 9.0188,C 0.2469,E1 8.862,E2 269.0896} C_DIS
LIN {X -137.6559,Y 0.7997,Z 171,A -179.1585,B 9.019,C 0.2409,E1 8.862,E2 270.6882} C_DIS
LIN {X -137.5937,Y 4.193,Z 171,A 179.3092,B 9.019,C 0.2387,E1 8.862,E2 272.2339} C_DIS
LIN {X -137.4131,Y 8.1959,Z 171,A 177.5308,B 9.0191,C 0.2357,E1 8.8624,E2 274.0244} C_DIS
LIN {X -137.0452,Y 12.9657,Z 171,A 175.5935,B 9.0193,C 0.229,E1 8.8628,E2 275.953} C_DIS
LIN {X -136.63,Y 16.7903,Z 171,A 174.0685,B 9.0194,C 0.2232,E1 8.8633,E2 277.4671} C_DIS
LIN {X -136.0794,Y 20.7818,Z 171,A 172.3113,B 9.0195,C 0.2196,E1 8.864,E2 279.2325} C_DIS
LIN {X -135.3835,Y 24.9238,Z 171,A 170.5903,B 9.0197,C 0.2142,E1 8.8648,E2 280.9485} C_DIS
LIN {X -134.6849,Y 28.4558,Z 171,A 169.1496,B 9.0197,C 0.209,E1 8.8656,E2 282.3805} C_DIS
LIN {X -133.9631,Y 31.6802,Z 171,A 167.5687,B 9.0197,C 0.2084,E1 8.8666,E2 283.9854} C_DIS
LIN {X -132.9524,Y 35.6803,Z 171,A 165.9145,B 9.0199,C 0.2025,E1 8.8678,E2 285.6301} C_DIS
LIN {X -131.9992,Y 39.0607,Z 171,A 164.4606,B 9.02,C 0.1983,E1 8.8689,E2 287.0815} C_DIS
LIN {X -131.0591,Y 42.1061,Z 171,A 163.1028,B 9.02,C 0.1951,E1 8.8701,E2 288.4418} C_DIS
LIN {X -130.0079,Y 45.2473,Z 171,A 161.718,B 9.0202,C 0.1914,E1 8.8713,E2 289.8258} C_DIS
LIN {X -128.805,Y 48.5664,Z 171,A 160.1796,B 9.0202,C 0.1885,E1 8.8728,E2 291.3712} C_DIS
LIN {X -127.5284,Y 51.8267,Z 171,A 158.698,B 9.0202,C 0.185,E1 8.8743,E2 292.8544} C_DIS
LIN {X -126.1932,Y 54.9979,Z 171,A 157.2295,B 9.0204,C 0.1817,E1 8.8759,E2 294.3259} C_DIS
LIN {X -124.8157,Y 58.0556,Z 171,A 155.8156,B 9.0204,C 0.1783,E1 8.8776,E2 295.7405} C_DIS
LIN {X -123.0239,Y 61.7659,Z 171,A 154.1258,B 9.0205,C 0.1734,E1 8.8797,E2 297.4254} C_DIS
LIN {X -121.6004,Y 64.5213,Z 171,A 151.6227,B 9.0202,C 0.1899,E1 8.8832,E2 300.0746} C_DIS
LIN {X -117.6996,Y 71.3913,Z 171,A 149.469,B 9.0207,C 0.163,E1 8.886,E2 302.0873} C_DIS
LIN {X -115.6362,Y 74.6876,Z 171,A 147.6989,B 9.0207,C 0.1615,E1 8.8887,E2 303.8743} C_DIS
LIN {X -113.1839,Y 78.3542,Z 171,A 145.8251,B 9.0208,C 0.1577,E1 8.8916,E2 305.7508} C_DIS
LIN {X -110.8938,Y 81.5625,Z 171,A 143.6582,B 9.0208,C 0.1626,E1 8.8953,E2 307.9802} C_DIS
LIN {X -107.8432,Y 85.5556,Z 171,A 142.0404,B 9.0209,C 0.1499,E1 8.898,E2 309.5382} C_DIS
LIN {X -104.977,Y 89.049,Z 171,A 140.154,B 9.021,C 0.1457,E1 8.9014,E2 311.4234} C_DIS
LIN {X -101.3036,Y 93.2065,Z 171,A 138.1221,B 9.0212,C 0.136,E1 8.9051,E2 313.419} C_DIS
LIN {X -99.2831,Y 95.3564,Z 171,A 136.6172,B 9.0212,C 0.1381,E1 8.9081,E2 314.9568} C_DIS
LIN {X -96.4658,Y 98.205,Z 171,A 134.8853,B 9.0212,C 0.1357,E1 8.9115,E2 316.6948} C_DIS
LIN {X -93.0203,Y 101.4748,Z 171,A 132.9535,B 9.0212,C 0.131,E1 8.9154,E2 318.6192} C_DIS
LIN {X -90.0859,Y 104.089,Z 171,A 131.2126,B 9.0212,C 0.1296,E1 8.9191,E2 320.3714} C_DIS
LIN {X -86.625,Y 106.9862,Z 171,A 129.3077,B 9.0212,C 0.1265,E1 8.9232,E2 322.2777} C_DIS
LIN {X -82.3162,Y 110.3355,Z 171,A 127.0415,B 9.0214,C 0.1224,E1 8.9282,E2 324.5412} C_DIS
LIN {X -78.7574,Y 112.9034,Z 171,A 125.2037,B 9.0214,C 0.1195,E1 8.9324,E2 326.3787} C_DIS
LIN {X -75.1407,Y 115.3421,Z 171,A 123.3058,B 9.0214,C 0.1179,E1 8.9368,E2 328.285} C_DIS
LIN {X -70.9436,Y 117.9703,Z 171,A 121.3181,B 9.0214,C 0.1135,E1 8.9415,E2 330.2619} C_DIS
LIN {X -66.4007,Y 120.5857,Z 171,A 119.2365,B 9.0215,C 0.1085,E1 8.9466,E2 332.3295} C_DIS
LIN {X -62.9151,Y 122.4389,Z 171,A 117.3585,B 9.0215,C 0.1104,E1 8.9513,E2 334.2347} C_DIS
LIN {X -59.0401,Y 124.3531,Z 171,A 115.6465,B 9.0215,C 0.1066,E1 8.9556,E2 335.9346} C_DIS
LIN {X -54.9511,Y 126.2134,Z 171,A 113.7423,B 9.0215,C 0.1049,E1 8.9604,E2 337.8415} C_DIS
LIN {X -51.2797,Y 127.7488,Z 171,A 112.1675,B 9.0216,C 0.1016,E1 8.9645,E2 339.4051} C_DIS
LIN {X -47.9208,Y 129.0469,Z 171,A 110.2611,B 9.0216,C 0.1074,E1 8.9696,E2 341.3599} C_DIS
LIN {X -44.2125,Y 130.3656,Z 171,A 108.8962,B 9.0216,C 0.1009,E1 8.9731,E2 342.6906} C_DIS
LIN {X -40.4908,Y 131.5671,Z 171,A 107.3753,B 9.0216,C 0.0974,E1 8.9771,E2 344.1971} C_DIS
LIN {X -37.0935,Y 132.5649,Z 171,A 105.8656,B 9.0216,C 0.0969,E1 8.9812,E2 345.7102} C_DIS
LIN {X -33.5681,Y 133.5015,Z 171,A 104.3541,B 9.0216,C 0.0956,E1 8.9852,E2 347.2199} C_DIS
LIN {X -30.2464,Y 134.2934,Z 171,A 102.927,B 9.0216,C 0.0948,E1 8.9891,E2 348.6468} C_DIS
LIN {X -27.0695,Y 134.9696,Z 171,A 101.583,B 9.0216,C 0.0938,E1 8.9928,E2 349.9889} C_DIS
LIN {X -22.9821,Y 135.7253,Z 171,A 99.5939,B 9.0216,C 0.0977,E1 8.9984,E2 352.0086} C_DIS
LIN {X -17.6253,Y 136.5242,Z 171,A 97.6262,B 9.0217,C 0.0914,E1 9.0037,E2 353.94} C_DIS
LIN {X -11.4473,Y 137.1803,Z 171,A 95.3312,B 9.0217,C 0.0851,E1 9.01,E2 356.198} C_DIS
LIN {X -4.2416,Y 137.5924,Z 171,A 92.1527,B 9.0217,C 0.0879,E1 9.0189,E2 359.3967} C_DIS
LIN {X 2.6091,Y 137.6328,Z 171,A 89.4103,B 9.0217,C 0.0857,E1 9.0265,E2 362.1246} C_DIS
LIN {X 9.6453,Y 137.3192,Z 171,A 86.1916,B 9.0217,C 0.0917,E1 9.0356,E2 365.3775} C_DIS
LIN {X 16.5112,Y 136.6633,Z 171,A 83.3062,B 9.0217,C 0.0927,E1 9.0436,E2 368.2637} C_DIS
LIN {X 22.036,Y 135.8831,Z 171,A 81.1089,B 9.0217,C 0.0912,E1 9.0496,E2 370.445} C_DIS
LIN {X 26.2061,Y 135.1399,Z 171,A 79.2785,B 9.0217,C 0.0934,E1 9.0547,E2 372.2831} C_DIS
LIN {X 29.3803,Y 134.4853,Z 171,A 77.5668,B 9.0217,C 0.1014,E1 9.0595,E2 374.0388} C_DIS
LIN {X 33.0614,Y 133.6301,Z 171,A 76.3665,B 9.0217,C 0.095,E1 9.0626,E2 375.1933} C_DIS
LIN {X 36.5141,Y 132.7269,Z 171,A 74.8133,B 9.0217,C 0.0975,E1 9.0668,E2 376.7545} C_DIS
LIN {X 40.3766,Y 131.6021,Z 171,A 73.1999,B 9.0217,C 0.0975,E1 9.0711,E2 378.3601} C_DIS
LIN {X 43.5144,Y 130.5981,Z 171,A 71.8599,B 9.0217,C 0.0981,E1 9.0747,E2 379.696} C_DIS
LIN {X 46.6407,Y 129.5145,Z 171,A 70.4142,B 9.0217,C 0.1008,E1 9.0785,E2 381.15} C_DIS
LIN {X 50.203,Y 128.1761,Z 171,A 68.871,B 9.0217,C 0.1016,E1 9.0825,E2 382.6881} C_DIS
LIN {X 53.4382,Y 126.8616,Z 171,A 67.4581,B 9.0216,C 0.1024,E1 9.0861,E2 384.0958} C_DIS
LIN {X 56.5853,Y 125.4895,Z 171,A 66.0339,B 9.0216,C 0.1039,E1 9.0898,E2 385.5195} C_DIS
LIN {X 59.7195,Y 124.0285,Z 171,A 64.6079,B 9.0216,C 0.1054,E1 9.0934,E2 386.9438} C_DIS
LIN {X 64.3245,Y 121.7038,Z 171,A 62.62,B 9.0216,C 0.1049,E1 9.0983,E2 388.9121} C_DIS
LIN {X 67.5458,Y 119.9477,Z 171,A 60.875,B 9.0215,C 0.1115,E1 9.1026,E2 390.6841} C_DIS
LIN {X 71.5379,Y 117.6109,Z 171,A 58.9618,B 9.0215,C 0.1141,E1 9.1072,E2 392.596} C_DIS
LIN {X 75.222,Y 115.2893,Z 171,A 57.1696,B 9.0215,C 0.1165,E1 9.1114,E2 394.3859} C_DIS
LIN {X 78.9661,Y 112.7581,Z 171,A 55.0922,B 9.0213,C 0.1236,E1 9.1162,E2 396.4877} C_DIS
LIN {X 81.6311,Y 110.8434,Z 171,A 54.1765,B 9.0214,C 0.1164,E1 9.1182,E2 397.3482} C_DIS
LIN {X 84.1447,Y 108.9477,Z 171,A 52.6198,B 9.0214,C 0.1239,E1 9.1217,E2 398.9356} C_DIS
LIN {X 87.7974,Y 106.0259,Z 171,A 50.7177,B 9.0213,C 0.1265,E1 9.1258,E2 400.8326} C_DIS
LIN {X 91.2004,Y 103.1133,Z 171,A 48.8967,B 9.0213,C 0.1291,E1 9.1296,E2 402.6488} C_DIS
LIN {X 94.3452,Y 100.2441,Z 171,A 46.9831,B 9.0212,C 0.1356,E1 9.1336,E2 404.5804} C_DIS
LIN {X 97.2997,Y 97.3796,Z 171,A 45.4238,B 9.0212,C 0.1357,E1 9.1366,E2 406.1214} C_DIS
LIN {X 102.0175,Y 92.4246,Z 171,A 42.8051,B 9.0212,C 0.1367,E1 9.1416,E2 408.7128} C_DIS
LIN {X 104.4084,Y 89.7149,Z 171,A 41.1574,B 9.0211,C 0.1431,E1 9.1447,E2 410.3788} C_DIS
LIN {X 107.1504,Y 86.4214,Z 171,A 39.3701,B 9.021,C 0.1471,E1 9.1478,E2 412.1674} C_DIS
LIN {X 109.9502,Y 82.8302,Z 171,A 37.5068,B 9.021,C 0.1507,E1 9.151,E2 414.0275} C_DIS
LIN {X 112.6465,Y 79.1246,Z 171,A 35.6104,B 9.0209,C 0.1549,E1 9.1541,E2 415.9236} C_DIS
LIN {X 115.1185,Y 75.483,Z 171,A 33.7905,B 9.0208,C 0.159,E1 9.1569,E2 417.7429} C_DIS
LIN {X 117.494,Y 71.7295,Z 171,A 31.9032,B 9.0207,C 0.1644,E1 9.1597,E2 419.636} C_DIS
LIN {X 119.9092,Y 67.6144,Z 171,A 30.0106,B 9.0207,C 0.1673,E1 9.1623,E2 421.5181} C_DIS
LIN {X 122.004,Y 63.7527,Z 171,A 28.3016,B 9.0207,C 0.1693,E1 9.1645,E2 423.2133} C_DIS
LIN {X 123.6385,Y 60.5229,Z 171,A 26.8125,B 9.0205,C 0.1728,E1 9.1664,E2 424.7011} C_DIS
LIN {X 125.2321,Y 57.1551,Z 171,A 25.2358,B 9.0205,C 0.1774,E1 9.1682,E2 426.2822} C_DIS
LIN {X 126.9578,Y 53.208,Z 171,A 23.421,B 9.0203,C 0.1826,E1 9.1702,E2 428.1007} C_DIS
LIN {X 128.2725,Y 49.9551,Z 171,A 22.0471,B 9.0203,C 0.1846,E1 9.1716,E2 429.4649} C_DIS
LIN {X 129.6314,Y 46.3164,Z 171,A 20.4987,B 9.0203,C 0.1874,E1 9.1731,E2 431.0059} C_DIS
LIN {X 130.9696,Y 42.3863,Z 171,A 18.7356,B 9.0201,C 0.193,E1 9.1747,E2 432.7747} C_DIS
LIN {X 132.149,Y 38.549,Z 171,A 17.1865,B 9.0201,C 0.1948,E1 9.1759,E2 434.3099} C_DIS
LIN {X 133.0382,Y 35.3586,Z 171,A 15.7791,B 9.02,C 0.1993,E1 9.177,E2 435.722} C_DIS
LIN {X 133.9186,Y 31.8649,Z 171,A 14.3132,B 9.02,C 0.2028,E1 9.1779,E2 437.1849} C_DIS
LIN {X 134.9065,Y 27.3796,Z 171,A 12.4612,B 9.0198,C 0.2068,E1 9.179,E2 439.031} C_DIS
LIN {X 135.5345,Y 24.0801,Z 171,A 11.0179,B 9.0198,C 0.2118,E1 9.1797,E2 440.4811} C_DIS
LIN {X 136.335,Y 19.0367,Z 171,A 9.0455,B 9.0196,C 0.2144,E1 9.1806,E2 442.4361} C_DIS
LIN {X 136.6979,Y 16.2209,Z 171,A 7.5237,B 9.0194,C 0.2256,E1 9.1811,E2 444.0016} C_DIS
LIN {X 137.0463,Y 12.9528,Z 171,A 6.5093,B 9.0194,C 0.2215,E1 9.1814,E2 444.9728} C_DIS
LIN {X 137.451,Y 7.5347,Z 171,A 4.0193,B 9.0192,C 0.2332,E1 9.1818,E2 447.4936} C_DIS
LIN {X 137.6475,Y 1.6751,Z 171,A 1.5474,B 9.019,C 0.241,E1 9.182,E2 449.9718} C_DIS
LIN {X 137.6481,Y -1.6863,Z 171,A 0.5515,B 9.0191,C 0.2359,E1 9.182,E2 450.9183} C_DIS
LIN {X 137.3528,Y -9.1756,Z 171,A -3.1491,B 9.0185,C 0.2582,E1 9.1814,E2 454.695} C_DIS
LIN {X 136.9692,Y -13.7464,Z 171,A -4.6395,B 9.0186,C 0.2542,E1 9.1811,E2 456.1347} C_DIS
LIN {X 136.5078,Y -17.7505,Z 171,A -6.6331,B 9.0183,C 0.2663,E1 9.1803,E2 458.1696} C_DIS
LIN {X 135.859,Y -22.1808,Z 171,A -8.2981,B 9.0183,C 0.2671,E1 9.1796,E2 459.8115} C_DIS
LIN {X 135.2588,Y -25.5841,Z 171,A -9.4954,B 9.0183,C 0.2658,E1 9.179,E2 460.98} C_DIS
LIN {X 134.4033,Y -29.7604,Z 171,A -11.3099,B 9.0181,C 0.2718,E1 9.1779,E2 462.8013} C_DIS
LIN {X 133.4416,Y -33.8044,Z 171,A -12.8742,B 9.0181,C 0.2729,E1 9.1769,E2 464.3464} C_DIS
LIN {X 132.5848,Y -37.0223,Z 171,A -14.5347,B 9.0178,C 0.2831,E1 9.1756,E2 466.043} C_DIS
LIN {X 131.5856,Y -40.4303,Z 171,A -15.6598,B 9.0178,C 0.2792,E1 9.1748,E2 467.1251} C_DIS
LIN {X 130.5166,Y -43.7592,Z 171,A -17.0982,B 9.0178,C 0.2829,E1 9.1735,E2 468.5629} C_DIS
LIN {X 129.2286,Y -47.4336,Z 171,A -18.9729,B 9.0175,C 0.2931,E1 9.1717,E2 470.4714} C_DIS
LIN {X 128.0845,Y -50.4389,Z 171,A -19.9686,B 9.0175,C 0.289,E1 9.1707,E2 471.4251} C_DIS
LIN {X 126.9414,Y -53.2472,Z 171,A -21.2508,B 9.0175,C 0.2929,E1 9.1694,E2 472.7112} C_DIS
LIN {X 125.3293,Y -56.9435,Z 171,A -23.4898,B 9.0169,C 0.3101,E1 9.1667,E2 475.0228} C_DIS
LIN {X 123.2317,Y -61.3475,Z 171,A -24.9105,B 9.0172,C 0.3017,E1 9.1651,E2 476.3686} C_DIS
LIN {X 121.7373,Y -64.2607,Z 171,A -26.2585,B 9.0171,C 0.3049,E1 9.1633,E2 477.7162} C_DIS
LIN {X 119.7552,Y -67.8875,Z 171,A -28.0046,B 9.0169,C 0.31,E1 9.1609,E2 479.4675} C_DIS
LIN {X 117.9068,Y -71.0485,Z 171,A -30.08,B 9.0163,C 0.3262,E1 9.1579,E2 481.6141} C_DIS
LIN {X 115.119,Y -75.4821,Z 171,A -31.5255,B 9.0167,C 0.3152,E1 9.1558,E2 482.969} C_DIS
LIN {X 113.2443,Y -78.2672,Z 171,A -33.0934,B 9.0165,C 0.3225,E1 9.1533,E2 484.5601} C_DIS
LIN {X 110.5859,Y -81.98,Z 171,A -34.8984,B 9.0164,C 0.3249,E1 9.1503,E2 486.3549} C_DIS
LIN {X 107.5931,Y -85.8699,Z 171,A -36.7004,B 9.0164,C 0.3243,E1 9.1473,E2 488.1283} C_DIS
LIN {X 105.6604,Y -88.2375,Z 171,A -38.2255,B 9.0161,C 0.3329,E1 9.1445,E2 489.687} C_DIS
LIN {X 102.57,Y -91.811,Z 171,A -39.9838,B 9.0161,C 0.3327,E1 9.1413,E2 491.4208} C_DIS
LIN {X 98.0439,Y -96.6301,Z 171,A -42.6173,B 9.016,C 0.3361,E1 9.1363,E2 494.0421} C_DIS
LIN {X 95.3,Y -99.3371,Z 171,A -44.7239,B 9.0154,C 0.3506,E1 9.132,E2 496.2142} C_DIS
LIN {X 92.5992,Y -101.8591,Z 171,A -45.6479,B 9.0158,C 0.3402,E1 9.1302,E2 497.0615} C_DIS
LIN {X 87.8436,Y -105.9876,Z 171,A -48.4657,B 9.0154,C 0.3498,E1 9.1242,E2 499.9071} C_DIS
LIN {X 84.7538,Y -108.4748,Z 171,A -50.8033,B 9.0147,C 0.3678,E1 9.1189,E2 502.3334} C_DIS
LIN {X 80.331,Y -111.7896,Z 171,A -52.5913,B 9.015,C 0.3609,E1 9.115,E2 504.0587} C_DIS
LIN {X 76.1388,Y -114.686,Z 171,A -54.5881,B 9.015,C 0.3618,E1 9.1104,E2 506.0416} C_DIS
LIN {X 72.3802,Y -117.0946,Z 171,A -56.5832,B 9.0147,C 0.3678,E1 9.1056,E2 508.0559} C_DIS
LIN {X 69.2771,Y -118.9566,Z 171,A -57.9406,B 9.0147,C 0.367,E1 9.1024,E2 509.3957} C_DIS
LIN {X 65.4041,Y -121.1291,Z 171,A -59.7384,B 9.0147,C 0.3687,E1 9.098,E2 511.1887} C_DIS
LIN {X 62.0027,Y -122.9033,Z 171,A -61.3534,B 9.0146,C 0.3714,E1 9.094,E2 512.8074} C_DIS
LIN {X 58.1451,Y -124.7743,Z 171,A -63.0711,B 9.0146,C 0.3724,E1 9.0897,E2 514.5179} C_DIS
LIN {X 52.92,Y -127.078,Z 171,A -65.3504,B 9.0146,C 0.3733,E1 9.0839,E2 516.7868} C_DIS
LIN {X 47.2422,Y -129.2976,Z 171,A -67.7873,B 9.0145,C 0.3741,E1 9.0776,E2 519.2129} C_DIS
LIN {X 41.7625,Y -131.1689,Z 171,A -70.2848,B 9.0143,C 0.3784,E1 9.0709,E2 521.7233} C_DIS
LIN {X 38.5135,Y -132.1594,Z 171,A -71.7071,B 9.0143,C 0.38,E1 9.0671,E2 523.1478} C_DIS
LIN {X 34.7604,Y -133.1977,Z 171,A -73.5749,B 9.014,C 0.3865,E1 9.062,E2 525.0482} C_DIS
LIN {X 29.6051,Y -134.4368,Z 171,A -75.6096,B 9.014,C 0.3847,E1 9.0565,E2 527.0625} C_DIS
LIN {X 25.4119,Y -135.2917,Z 171,A -77.2396,B 9.0141,C 0.3827,E1 9.0521,E2 528.6743} C_DIS
LIN {X 22.2813,Y -135.8422,Z 171,A -78.5967,B 9.0141,C 0.3842,E1 9.0483,E2 530.0366} C_DIS
LIN {X 16.0993,Y -136.7124,Z 171,A -80.907,B 9.0142,C 0.3797,E1 9.042,E2 532.3116} C_DIS
LIN {X 13.0118,Y -137.0407,Z 171,A -82.9106,B 9.0136,C 0.3947,E1 9.0362,E2 534.4066} C_DIS
LIN {X 8.8884,Y -137.3704,Z 171,A -84.0309,B 9.0141,C 0.3831,E1 9.0333,E2 535.4513} C_DIS
LIN {X 5.5698,Y -137.5445,Z 171,A -85.5872,B 9.0139,C 0.387,E1 9.0289,E2 537.0305} C_DIS
LIN {X 1.9047,Y -137.6445,Z 171,A -87.0748,B 9.0139,C 0.3865,E1 9.0247,E2 538.514} C_DIS
LIN {X 1.9047,Y -137.6445,Z 171,A -87.0748,B 9.0139,C 0.3865,E1 9.0247,E2 538.514} C_DIS
Enddeposition()
LIN {X 1.0061,Y -138.56,Z 171,A -87.0796,B 8.9741,C 0.3852,E1 8.9848,E2 538.5171} C_DIS
Startdeposition()
$VEL.CP = VEL_PRINT
LIN {X 4.1254,Y -138.5063,Z 171,A -85.4706,B 8.9744,C 0.3785,E1 8.9895,E2 536.8662} C_DIS
LIN {X 8.3167,Y -138.3177,Z 171,A -83.7961,B 8.9744,C 0.3793,E1 8.9941,E2 535.1986} C_DIS
LIN {X 12.5875,Y -137.996,Z 171,A -81.912,B 8.9744,C 0.3763,E1 8.9994,E2 533.2989} C_DIS
LIN {X 16.6347,Y -137.5653,Z 171,A -79.6845,B 8.975,C 0.3641,E1 9.0058,E2 530.999} C_DIS
LIN {X 21.8788,Y -136.83,Z 171,A -78.2304,B 8.9744,C 0.3783,E1 9.0095,E2 529.6399} C_DIS
LIN {X 25.6073,Y -136.1811,Z 171,A -76.5416,B 8.9746,C 0.3747,E1 9.0142,E2 527.9339} C_DIS
LIN {X 29.2349,Y -135.448,Z 171,A -75.0661,B 8.9746,C 0.3747,E1 9.0182,E2 526.4646} C_DIS
LIN {X 35.0835,Y -134.0537,Z 171,A -72.5132,B 8.9746,C 0.3714,E1 9.0252,E2 523.9014} C_DIS
LIN {X 38.7778,Y -133.0306,Z 171,A -71.002,B 8.9746,C 0.3714,E1 9.0292,E2 522.3986} C_DIS
LIN {X 41.9902,Y -132.0518,Z 171,A -69.6304,B 8.9747,C 0.3705,E1 9.0329,E2 521.0282} C_DIS
LIN {X 45.3589,Y -130.9327,Z 171,A -68.097,B 8.9748,C 0.3676,E1 9.0369,E2 519.4852} C_DIS
LIN {X 50.8538,Y -128.8998,Z 171,A -65.6353,B 8.975,C 0.364,E1 9.0434,E2 517.0165} C_DIS
LIN {X 54.8062,Y -127.2678,Z 171,A -63.7883,B 8.9751,C 0.36,E1 9.0482,E2 515.1578} C_DIS
LIN {X 59.1814,Y -125.2945,Z 171,A -62.026,B 8.9751,C 0.3622,E1 9.0526,E2 513.4229} C_DIS
LIN {X 62.684,Y -123.578,Z 171,A -60.4199,B 8.9751,C 0.3601,E1 9.0566,E2 511.8162} C_DIS
LIN {X 65.9959,Y -121.8443,Z 171,A -58.7844,B 8.9753,C 0.3559,E1 9.0606,E2 510.1679} C_DIS
LIN {X 69.4457,Y -119.9109,Z 171,A -56.5679,B 8.9759,C 0.3405,E1 9.0662,E2 507.8736} C_DIS
LIN {X 74.3244,Y -116.9504,Z 171,A -54.8406,B 8.9755,C 0.3507,E1 9.0701,E2 506.2273} C_DIS
LIN {X 78.0578,Y -114.4923,Z 171,A -52.5799,B 8.976,C 0.3383,E1 9.0754,E2 503.9109} C_DIS
LIN {X 81.8565,Y -111.8074,Z 171,A -50.7464,B 8.976,C 0.3369,E1 9.0795,E2 502.0873} C_DIS
LIN {X 85.295,Y -109.2073,Z 171,A -49.3113,B 8.9759,C 0.3413,E1 9.0826,E2 500.6961} C_DIS
LIN {X 88.0861,Y -106.9687,Z 171,A -47.2566,B 8.9765,C 0.3255,E1 9.0872,E2 498.5646} C_DIS
LIN {X 92.4238,Y -103.2433,Z 171,A -45.6596,B 8.976,C 0.3381,E1 9.0904,E2 497.0658} C_DIS
LIN {X 96.275,Y -99.6618,Z 171,A -43.3927,B 8.9762,C 0.3315,E1 9.095,E2 494.7847} C_DIS
LIN {X 98.6556,Y -97.3065,Z 171,A -41.4621,B 8.9768,C 0.3162,E1 9.0989,E2 492.7814} C_DIS
LIN {X 102.3726,Y -93.3878,Z 171,A -39.9737,B 8.9764,C 0.3281,E1 9.1015,E2 491.3881} C_DIS
LIN {X 107.3104,Y -87.6687,Z 171,A -36.9512,B 8.9765,C 0.3234,E1 9.107,E2 488.3758} C_DIS
LIN {X 110.953,Y -83.011,Z 171,A -34.192,B 8.977,C 0.3104,E1 9.1118,E2 485.5733} C_DIS
LIN {X 113.9635,Y -78.8276,Z 171,A -32.2041,B 8.977,C 0.3085,E1 9.1149,E2 483.6018} C_DIS
LIN {X 115.7798,Y -76.1339,Z 171,A -30.6587,B 8.9773,C 0.3006,E1 9.1174,E2 482.0288} C_DIS
LIN {X 117.7176,Y -73.1021,Z 171,A -29.4225,B 8.9773,C 0.3026,E1 9.1191,E2 480.8237} C_DIS
LIN {X 119.8898,Y -69.4822,Z 171,A -27.7324,B 8.9773,C 0.2994,E1 9.1215,E2 479.1391} C_DIS
LIN {X 122.0855,Y -65.5475,Z 171,A -26.0204,B 8.9774,C 0.2981,E1 9.1238,E2 477.4447} C_DIS
LIN {X 123.7619,Y -62.3227,Z 171,A -24.4995,B 8.9775,C 0.2937,E1 9.1258,E2 475.9198} C_DIS
LIN {X 127.9477,Y -53.1997,Z 171,A -20.7915,B 8.9775,C 0.2928,E1 9.13,E2 472.2649} C_DIS
LIN {X 130.1025,Y -47.6937,Z 171,A -17.8935,B 8.9781,C 0.2757,E1 9.133,E2 469.3063} C_DIS
LIN {X 131.3305,Y -44.1961,Z 171,A -16.5107,B 8.9781,C 0.2749,E1 9.1342,E2 467.9412} C_DIS
LIN {X 132.4354,Y -40.7644,Z 171,A -14.4651,B 8.9786,C 0.2578,E1 9.136,E2 465.822} C_DIS
LIN {X 133.7763,Y -36.1239,Z 171,A -13.0647,B 8.9784,C 0.2661,E1 9.1369,E2 464.4971} C_DIS
LIN {X 134.6825,Y -32.5801,Z 171,A -11.5251,B 8.9785,C 0.2611,E1 9.138,E2 462.9524} C_DIS
LIN {X 135.5826,Y -28.6117,Z 171,A -9.3671,B 8.979,C 0.2453,E1 9.1393,E2 460.7311} C_DIS
LIN {X 136.4703,Y -24.0186,Z 171,A -8.0892,B 8.9787,C 0.255,E1 9.1399,E2 459.5363} C_DIS
LIN {X 136.9973,Y -20.8033,Z 171,A -6.5691,B 8.9789,C 0.2471,E1 9.1405,E2 457.9925} C_DIS
LIN {X 137.5679,Y -16.6134,Z 171,A -5.1642,B 8.9789,C 0.25,E1 9.141,E2 456.6301} C_DIS
LIN {X 138.2136,Y -9.8969,Z 171,A -2.3366,B 8.9791,C 0.2411,E1 9.1418,E2 453.7952} C_DIS
LIN {X 138.519,Y -3.6668,Z 171,A 0.3769,B 8.9794,C 0.2305,E1 9.1421,E2 451.0621} C_DIS
LIN {X 138.5675,Y -0.6222,Z 171,A 2.1002,B 8.9797,C 0.216,E1 9.1421,E2 449.2777} C_DIS
LIN {X 138.5097,Y 4.0022,Z 171,A 4.0556,B 8.9799,C 0.2095,E1 9.1419,E2 447.315} C_DIS
LIN {X 138.2634,Y 9.1986,Z 171,A 5.6466,B 8.9797,C 0.2163,E1 9.1417,E2 445.7944} C_DIS
LIN {X 137.9844,Y 12.7075,Z 171,A 7.7714,B 8.9802,C 0.1965,E1 9.1411,E2 443.5818} C_DIS
LIN {X 137.2931,Y 18.7638,Z 171,A 9.4371,B 8.9799,C 0.2091,E1 9.1405,E2 442.0244} C_DIS
LIN {X 136.5349,Y 23.6574,Z 171,A 11.6031,B 8.9801,C 0.2006,E1 9.1396,E2 439.8415} C_DIS
LIN {X 135.9726,Y 26.698,Z 171,A 13.2057,B 8.9803,C 0.1895,E1 9.1387,E2 438.1962} C_DIS
LIN {X 135.1089,Y 30.7645,Z 171,A 14.4469,B 8.9802,C 0.1956,E1 9.138,E2 437.0149} C_DIS
LIN {X 134.2582,Y 34.2872,Z 171,A 15.928,B 8.9802,C 0.1918,E1 9.137,E2 435.5348} C_DIS
LIN {X 133.1302,Y 38.4377,Z 171,A 17.7388,B 8.9804,C 0.1861,E1 9.1356,E2 433.7186} C_DIS
LIN {X 132.0843,Y 41.8883,Z 171,A 19.0987,B 8.9804,C 0.185,E1 9.1345,E2 432.3743} C_DIS
LIN {X 131.0613,Y 44.988,Z 171,A 20.5313,B 8.9805,C 0.1794,E1 9.1332,E2 430.9301} C_DIS
LIN {X 129.7414,Y 48.6617,Z 171,A 22.0728,B 8.9805,C 0.1767,E1 9.1317,E2 429.3967} C_DIS
LIN {X 128.7072,Y 51.3372,Z 171,A 23.6662,B 8.9808,C 0.1643,E1 9.13,E2 427.7503} C_DIS
LIN {X 127.1126,Y 55.1654,Z 171,A 24.9411,B 8.9808,C 0.1697,E1 9.1287,E2 426.5306} C_DIS
LIN {X 125.5668,Y 58.6002,Z 171,A 26.5104,B 8.9808,C 0.1654,E1 9.1268,E2 424.9588} C_DIS
LIN {X 123.6537,Y 62.5352,Z 171,A 28.2096,B 8.9808,C 0.1632,E1 9.1247,E2 423.2725} C_DIS
LIN {X 121.8818,Y 65.9266,Z 171,A 29.8976,B 8.981,C 0.1568,E1 9.1225,E2 421.5701} C_DIS
LIN {X 119.7652,Y 69.6975,Z 171,A 31.9815,B 8.9811,C 0.1457,E1 9.1195,E2 419.4474} C_DIS
LIN {X 117.6546,Y 73.2033,Z 171,A 33.2963,B 8.9811,C 0.1501,E1 9.1177,E2 418.1798} C_DIS
LIN {X 115.1627,Y 77.0643,Z 171,A 35.1961,B 8.9811,C 0.1455,E1 9.1148,E2 416.279} C_DIS
LIN {X 112.5619,Y 80.8159,Z 171,A 37.054,B 8.9812,C 0.1417,E1 9.1118,E2 414.424} C_DIS
LIN {X 109.8928,Y 84.4097,Z 171,A 38.8818,B 8.9812,C 0.138,E1 9.1087,E2 412.5983} C_DIS
LIN {X 107.048,Y 87.9898,Z 171,A 40.7586,B 8.9813,C 0.1341,E1 9.1054,E2 410.7224} C_DIS
LIN {X 104.1289,Y 91.4258,Z 171,A 42.4846,B 8.9813,C 0.1331,E1 9.1023,E2 409.0131} C_DIS
LIN {X 99.9613,Y 95.9643,Z 171,A 45.2577,B 8.9815,C 0.1228,E1 9.0969,E2 406.2107} C_DIS
LIN {X 97.5612,Y 98.4031,Z 171,A 46.4573,B 8.9815,C 0.1247,E1 9.0946,E2 405.0378} C_DIS
LIN {X 93.8343,Y 101.963,Z 171,A 48.615,B 8.9815,C 0.1199,E1 9.0902,E2 402.8761} C_DIS
LIN {X 90.3107,Y 105.0968,Z 171,A 50.5324,B 8.9815,C 0.1169,E1 9.0862,E2 400.9623} C_DIS
LIN {X 86.8344,Y 107.9868,Z 171,A 52.3804,B 8.9815,C 0.114,E1 9.0822,E2 399.1165} C_DIS
LIN {X 83.2057,Y 110.8073,Z 171,A 54.0811,B 8.9815,C 0.115,E1 9.0785,E2 397.4406} C_DIS
LIN {X 77.4112,Y 114.9301,Z 171,A 57.1614,B 8.9817,C 0.1072,E1 9.0714,E2 394.3424} C_DIS
LIN {X 73.7531,Y 117.311,Z 171,A 58.7972,B 8.9817,C 0.108,E1 9.0676,E2 392.7276} C_DIS
LIN {X 70.4001,Y 119.3533,Z 171,A 60.6053,B 8.9817,C 0.1017,E1 9.0632,E2 390.8962} C_DIS
LIN {X 66.37,Y 121.6402,Z 171,A 62.3761,B 8.9817,C 0.1021,E1 9.059,E2 389.1436} C_DIS
LIN {X 58.9547,Y 125.4027,Z 171,A 65.9466,B 8.9818,C 0.095,E1 9.05,E2 385.5567} C_DIS
LIN {X 55.4947,Y 126.9702,Z 171,A 67.2509,B 8.9818,C 0.0988,E1 9.0467,E2 384.2858} C_DIS
LIN {X 51.3185,Y 128.7147,Z 171,A 69.3271,B 8.9818,C 0.0925,E1 9.0413,E2 382.184} C_DIS
LIN {X 47.4066,Y 130.206,Z 171,A 70.9924,B 8.9818,C 0.0922,E1 9.037,E2 380.5271} C_DIS
LIN {X 43.9968,Y 131.3969,Z 171,A 72.4217,B 8.9818,C 0.0922,E1 9.0332,E2 379.106} C_DIS
LIN {X 40.7732,Y 132.4327,Z 171,A 73.7919,B 8.9818,C 0.0915,E1 9.0296,E2 377.7398} C_DIS
LIN {X 37.521,Y 133.3906,Z 171,A 75.1765,B 8.9818,C 0.0908,E1 9.0259,E2 376.3576} C_DIS
LIN {X 33.9915,Y 134.3333,Z 171,A 77.7396,B 8.9821,C 0.0682,E1 9.0186,E2 373.662} C_DIS
LIN {X 26.8137,Y 135.9505,Z 171,A 79.8908,B 8.9819,C 0.0847,E1 9.013,E2 371.6245} C_DIS
LIN {X 23.0624,Y 136.6348,Z 171,A 81.8632,B 8.9819,C 0.076,E1 9.0074,E2 369.6027} C_DIS
LIN {X 18.4532,Y 137.3338,Z 171,A 83.1947,B 8.9819,C 0.0872,E1 9.004,E2 368.3467} C_DIS
LIN {X 11.9365,Y 138.0525,Z 171,A 85.974,B 8.9819,C 0.0851,E1 8.9962,E2 365.5599} C_DIS
LIN {X 9.1616,Y 138.2657,Z 171,A 87.6838,B 8.982,C 0.0738,E1 8.9913,E2 363.7805} C_DIS
LIN {X 4.3659,Y 138.4993,Z 171,A 89.2006,B 8.982,C 0.0829,E1 8.9872,E2 362.3235} C_DIS
LIN {X -0.7088,Y 138.5657,Z 171,A 91.2311,B 8.982,C 0.0843,E1 8.9815,E2 360.3023} C_DIS
LIN {X -4.6783,Y 138.4903,Z 171,A 93.5726,B 8.982,C 0.0708,E1 8.9748,E2 357.8739} C_DIS
LIN {X -10.3115,Y 138.1833,Z 171,A 94.971,B 8.9819,C 0.0895,E1 8.9712,E2 356.5937} C_DIS
LIN {X -18.0601,Y 137.3853,Z 171,A 98.0622,B 8.9819,C 0.093,E1 8.9627,E2 353.5207} C_DIS
LIN {X -20.3148,Y 137.0704,Z 171,A 99.763,B 8.9819,C 0.079,E1 8.9577,E2 351.7259} C_DIS
LIN {X -24.24,Y 136.4306,Z 171,A 101.1327,B 8.9819,C 0.0851,E1 8.954,E2 350.3915} C_DIS
LIN {X -29.0063,Y 135.4974,Z 171,A 103.0425,B 8.9819,C 0.0881,E1 8.9488,E2 348.4953} C_DIS
LIN {X -32.3948,Y 134.7272,Z 171,A 104.3372,B 8.9819,C 0.0918,E1 8.9454,E2 347.2192} C_DIS
LIN {X -35.4614,Y 133.9529,Z 171,A 105.8177,B 8.9819,C 0.0895,E1 8.9413,E2 345.7182} C_DIS
LIN {X -38.9526,Y 132.9794,Z 171,A 107.2797,B 8.9819,C 0.0914,E1 8.9374,E2 344.2617} C_DIS
LIN {X -42.1522,Y 132,Z 171,A 108.6205,B 8.9819,C 0.0935,E1 8.9338,E2 342.9272} C_DIS
LIN {X -47.4249,Y 130.1994,Z 171,A 111.1629,B 8.9819,C 0.0913,E1 8.9271,E2 340.3568} C_DIS
LIN {X -51.5692,Y 128.6137,Z 171,A 112.7931,B 8.9818,C 0.0971,E1 8.9229,E2 338.7535} C_DIS
LIN {X -54.7465,Y 127.2937,Z 171,A 114.2151,B 8.9818,C 0.0987,E1 8.9192,E2 337.3327} C_DIS
LIN {X -57.6992,Y 125.9835,Z 171,A 115.4685,B 8.9818,C 0.1018,E1 8.9161,E2 336.0906} C_DIS
LIN {X -62.0074,Y 123.9212,Z 171,A 117.7426,B 8.9818,C 0.099,E1 8.9103,E2 333.7809} C_DIS
LIN {X -65.9122,Y 121.8895,Z 171,A 119.337,B 8.9817,C 0.1056,E1 8.9064,E2 332.2163} C_DIS
LIN {X -71.7317,Y 118.5576,Z 171,A 122.197,B 8.9817,C 0.1081,E1 8.8995,E2 329.3478} C_DIS
LIN {X -75.7825,Y 116.0107,Z 171,A 124.3294,B 8.9817,C 0.1085,E1 8.8944,E2 327.198} C_DIS
LIN {X -79.5627,Y 113.4515,Z 171,A 126.248,B 8.9817,C 0.1111,E1 8.89,E2 325.2773} C_DIS
LIN {X -82.1755,Y 111.573,Z 171,A 128.138,B 8.9817,C 0.1035,E1 8.8856,E2 323.3183} C_DIS
LIN {X -86.4065,Y 108.3294,Z 171,A 129.7778,B 8.9815,C 0.1175,E1 8.8822,E2 321.7515} C_DIS
LIN {X -89.817,Y 105.5189,Z 171,A 131.6248,B 8.9815,C 0.1206,E1 8.8782,E2 319.9038} C_DIS
LIN {X -93.8222,Y 101.9741,Z 171,A 134.1815,B 8.9815,C 0.119,E1 8.8729,E2 317.306} C_DIS
LIN {X -96.675,Y 99.2746,Z 171,A 135.5223,B 8.9815,C 0.1272,E1 8.8702,E2 316.0023} C_DIS
LIN {X -99.817,Y 96.1147,Z 171,A 137.2984,B 8.9813,C 0.1322,E1 8.8668,E2 314.2363} C_DIS
LIN {X -105.0814,Y 90.3286,Z 171,A 140.6468,B 8.9813,C 0.1374,E1 8.8605,E2 310.877} C_DIS
LIN {X -108.0261,Y 86.7857,Z 171,A 142.6117,B 8.9813,C 0.1407,E1 8.857,E2 308.9065} C_DIS
LIN {X -111.3598,Y 82.4649,Z 171,A 144.89,B 8.9811,C 0.1456,E1 8.8532,E2 306.6278} C_DIS
LIN {X -114.05,Y 78.7023,Z 171,A 146.8284,B 8.9811,C 0.1497,E1 8.8501,E2 304.6882} C_DIS
LIN {X -116.3375,Y 75.2792,Z 171,A 148.8163,B 8.9811,C 0.149,E1 8.847,E2 302.6661} C_DIS
LIN {X -118.3308,Y 72.1063,Z 171,A 149.894,B 8.9809,C 0.1609,E1 8.8455,E2 301.6492} C_DIS
LIN {X -121.3875,Y 66.832,Z 171,A 152.6885,B 8.9809,C 0.1627,E1 8.8416,E2 298.8231} C_DIS
LIN {X -123.3021,Y 63.2259,Z 171,A 154.3128,B 8.9807,C 0.1681,E1 8.8395,E2 297.2085} C_DIS
LIN {X -124.7773,Y 60.2639,Z 171,A 155.7125,B 8.9807,C 0.1712,E1 8.8378,E2 295.8063} C_DIS
LIN {X -126.3422,Y 56.9083,Z 171,A 157.2022,B 8.9806,C 0.176,E1 8.8361,E2 294.3233} C_DIS
LIN {X -127.7301,Y 53.7207,Z 171,A 158.6903,B 8.9806,C 0.179,E1 8.8344,E2 292.8304} C_DIS
LIN {X -129.0772,Y 50.3974,Z 171,A 160.1481,B 8.9805,C 0.1834,E1 8.8329,E2 291.3772} C_DIS
LIN {X -130.2413,Y 47.3087,Z 171,A 161.5337,B 8.9804,C 0.1868,E1 8.8316,E2 289.9904} C_DIS
LIN {X -131.3897,Y 44.0184,Z 171,A 163.0051,B 8.9804,C 0.1903,E1 8.8303,E2 288.5167} C_DIS
LIN {X -132.4062,Y 40.8597,Z 171,A 164.3653,B 8.9802,C 0.1943,E1 8.8291,E2 287.1595} C_DIS
LIN {X -133.3898,Y 37.524,Z 171,A 165.9227,B 8.9802,C 0.1964,E1 8.8279,E2 285.5885} C_DIS
LIN {X -134.2354,Y 34.377,Z 171,A 167.2922,B 8.9802,C 0.1998,E1 8.8269,E2 284.2176} C_DIS
LIN {X -135.0671,Y 30.9474,Z 171,A 168.7298,B 8.98,C 0.2043,E1 8.826,E2 282.7842} C_DIS
LIN {X -136.2557,Y 25.2144,Z 171,A 171.3987,B 8.98,C 0.2071,E1 8.8245,E2 280.0866} C_DIS
LIN {X -136.9363,Y 21.1974,Z 171,A 172.9347,B 8.9798,C 0.2144,E1 8.8239,E2 278.5709} C_DIS
LIN {X -137.5002,Y 17.1804,Z 171,A 174.6026,B 8.9797,C 0.2194,E1 8.8233,E2 276.906} C_DIS
LIN {X -138.0033,Y 12.5113,Z 171,A 176.6962,B 8.9796,C 0.2225,E1 8.8227,E2 274.795} C_DIS
LIN {X -138.4202,Y 6.4095,Z 171,A 179.2968,B 8.9794,C 0.2286,E1 8.8222,E2 272.1878} C_DIS
LIN {X -138.56,Y 1.5988,Z 171,A -178.4272,B 8.9794,C 0.2297,E1 8.8222,E2 269.8774} C_DIS
LIN {X -138.5537,Y -1.981,Z 171,A -176.9038,B 8.9794,C 0.2332,E1 8.8222,E2 268.3499} C_DIS
LIN {X -138.4476,Y -5.7741,Z 171,A -175.6292,B 8.9791,C 0.2427,E1 8.8223,E2 267.1142} C_DIS
LIN {X -138.2119,Y -9.9205,Z 171,A -173.9062,B 8.9789,C 0.2475,E1 8.8226,E2 265.392} C_DIS
LIN {X -137.7096,Y -15.4048,Z 171,A -171.5568,B 8.9788,C 0.2529,E1 8.8233,E2 263.0355} C_DIS
LIN {X -137.1989,Y -19.4262,Z 171,A -169.93,B 8.9786,C 0.2585,E1 8.8239,E2 261.4163} C_DIS
LIN {X -136.6843,Y -22.7655,Z 171,A -168.5664,B 8.9785,C 0.2631,E1 8.8245,E2 260.0581} C_DIS
LIN {X -136.1214,Y -25.9198,Z 171,A -167.1714,B 8.9785,C 0.2657,E1 8.8252,E2 258.6553} C_DIS
LIN {X -135.4759,Y -29.1058,Z 171,A -165.8085,B 8.9783,C 0.2691,E1 8.826,E2 257.2911} C_DIS
LIN {X -134.7358,Y -32.359,Z 171,A -164.377,B 8.9783,C 0.2721,E1 8.8269,E2 255.8542} C_DIS
LIN {X -133.8026,Y -36.0251,Z 171,A -162.7717,B 8.9781,C 0.2758,E1 8.828,E2 254.2448} C_DIS
LIN {X -132.5765,Y -40.3035,Z 171,A -160.9781,B 8.9779,C 0.2817,E1 8.8294,E2 252.4586} C_DIS
LIN {X -131.3003,Y -44.287,Z 171,A -158.7694,B 8.978,C 0.2782,E1 8.8314,E2 250.1901} C_DIS
LIN {X -129.9879,Y -48.0037,Z 171,A -157.5415,B 8.9777,C 0.2895,E1 8.8326,E2 249.0147} C_DIS
LIN {X -128.2955,Y -52.3584,Z 171,A -155.4217,B 8.9777,C 0.2914,E1 8.8348,E2 246.8723} C_DIS
LIN {X -126.6659,Y -56.1847,Z 171,A -153.7869,B 8.9774,C 0.2974,E1 8.8366,E2 245.2495} C_DIS
LIN {X -125.1529,Y -59.4778,Z 171,A -152.3218,B 8.9773,C 0.3018,E1 8.8383,E2 243.7896} C_DIS
LIN {X -123.6305,Y -62.5809,Z 171,A -150.8748,B 8.9772,C 0.3052,E1 8.8401,E2 242.3413} C_DIS
LIN {X -121.8379,Y -66.0067,Z 171,A -149.0884,B 8.9772,C 0.306,E1 8.8425,E2 240.5319} C_DIS
LIN {X -119.9078,Y -69.4511,Z 171,A -147.4888,B 8.977,C 0.3106,E1 8.8447,E2 238.9375} C_DIS
LIN {X -117.5344,Y -73.3964,Z 171,A -145.5574,B 8.9768,C 0.3147,E1 8.8475,E2 237.0036} C_DIS
LIN {X -115.045,Y -77.2406,Z 171,A -143.6218,B 8.9768,C 0.3185,E1 8.8505,E2 235.0637} C_DIS
LIN {X -112.488,Y -80.9194,Z 171,A -141.7157,B 8.9766,C 0.3218,E1 8.8536,E2 233.1515} C_DIS
LIN {X -109.7326,Y -84.6179,Z 171,A -139.788,B 8.9764,C 0.3257,E1 8.8568,E2 231.222} C_DIS
LIN {X -106.8964,Y -88.1735,Z 171,A -137.8985,B 8.9764,C 0.3297,E1 8.8602,E2 229.3323} C_DIS
LIN {X -104.3577,Y -91.1636,Z 171,A -135.7984,B 8.9764,C 0.3246,E1 8.8641,E2 227.1711} C_DIS
LIN {X -101.1513,Y -94.7094,Z 171,A -134.2466,B 8.9761,C 0.3363,E1 8.867,E2 225.6749} C_DIS
LIN {X -98.843,Y -97.1154,Z 171,A -132.69,B 8.9761,C 0.3358,E1 8.8701,E2 224.0958} C_DIS
LIN {X -96.5578,Y -99.388,Z 171,A -131.4995,B 8.9759,C 0.341,E1 8.8724,E2 222.9241} C_DIS
LIN {X -93.2154,Y -102.5291,Z 171,A -129.604,B 8.9758,C 0.3446,E1 8.8763,E2 221.0293} C_DIS
LIN {X -89.9198,Y -105.4315,Z 171,A -127.7658,B 8.9756,C 0.3475,E1 8.8802,E2 219.1887} C_DIS
LIN {X -86.525,Y -108.2351,Z 171,A -125.91,B 8.9756,C 0.35,E1 8.8842,E2 217.3288} C_DIS
LIN {X -80.7499,Y -112.6091,Z 171,A -122.914,B 8.9754,C 0.3549,E1 8.8909,E2 214.3334} C_DIS
LIN {X -77.1597,Y -115.099,Z 171,A -121.0639,B 8.9753,C 0.3569,E1 8.8952,E2 212.4778} C_DIS
LIN {X -73.199,Y -117.6573,Z 171,A -119.1235,B 8.9752,C 0.3599,E1 8.8998,E2 210.5389} C_DIS
LIN {X -69.1917,Y -120.0579,Z 171,A -117.2497,B 8.975,C 0.3637,E1 8.9043,E2 208.6727} C_DIS
LIN {X -62.1459,Y -123.852,Z 171,A -113.8432,B 8.975,C 0.366,E1 8.9127,E2 205.2537} C_DIS
LIN {X -58.4824,Y -125.6213,Z 171,A -112.2832,B 8.9747,C 0.3702,E1 8.9166,E2 203.7094} C_DIS
LIN {X -54.2991,Y -127.4871,Z 171,A -110.2257,B 8.9747,C 0.3691,E1 8.9219,E2 201.6307} C_DIS
LIN {X -50.5366,Y -129.0231,Z 171,A -108.6392,B 8.9747,C 0.3725,E1 8.926,E2 200.0563} C_DIS
LIN {X -47.1799,Y -130.2877,Z 171,A -107.1635,B 8.9746,C 0.374,E1 8.9299,E2 198.5813} C_DIS
LIN {X -43.9749,Y -131.4042,Z 171,A -105.756,B 8.9746,C 0.3751,E1 8.9336,E2 197.1731} C_DIS
LIN {X -40.7521,Y -132.4392,Z 171,A -104.382,B 8.9745,C 0.3766,E1 8.9372,E2 195.8021} C_DIS
LIN {X -37.6019,Y -133.368,Z 171,A -103.1356,B 8.9743,C 0.3797,E1 8.9405,E2 194.5699} C_DIS
LIN {X -28.6396,Y -135.5766,Z 171,A -99.0432,B 8.9745,C 0.3765,E1 8.9518,E2 190.4413} C_DIS
LIN {X -24.4328,Y -136.3961,Z 171,A -97.0387,B 8.9746,C 0.3726,E1 8.9573,E2 188.406} C_DIS
LIN {X -20.9271,Y -136.9781,Z 171,A -96.1158,B 8.9742,C 0.384,E1 8.9597,E2 187.5537} C_DIS
LIN {X -17.7928,Y -137.4203,Z 171,A -94.4524,B 8.9744,C 0.3773,E1 8.9644,E2 185.8437} C_DIS
LIN {X -13.4913,Y -137.9092,Z 171,A -92.7767,B 8.9744,C 0.3799,E1 8.969,E2 184.1823} C_DIS
LIN {X -10.0055,Y -138.2057,Z 171,A -91.3306,B 8.9744,C 0.38,E1 8.9731,E2 182.7357} C_DIS
LIN {X -5.9017,Y -138.4426,Z 171,A -89.6401,B 8.9744,C 0.3803,E1 8.9778,E2 181.0456} C_DIS
LIN {X -2.0994,Y -138.5517,Z 171,A -88.0639,B 8.9744,C 0.3801,E1 8.9822,E2 179.4683} C_DIS
LIN {X 1.0061,Y -138.56,Z 171,A -87.075,B 8.9741,C 0.3859,E1 8.9849,E2 178.517} C_DIS
Enddeposition()
LIN {X 1.0061,Y -138.56,Z 171,A -87.075,B 8.9741,C 0.3859,E1 8.9849,E2 178.517} C_DIS
Startdeposition()
$VEL.CP = VEL_PRINT
LIN {X -1.5644,Y -139.471,Z 171,A -88.5351,B 8.8339,C 0.4022,E1 8.8411,E2 180.105} C_DIS
LIN {X -5.5656,Y -139.3667,Z 171,A -90.0246,B 8.834,C 0.3991,E1 8.8369,E2 181.575} C_DIS
LIN {X -8.9579,Y -139.1903,Z 171,A -91.5082,B 8.834,C 0.4008,E1 8.8328,E2 183.0707} C_DIS
LIN {X -13.2144,Y -138.8503,Z 171,A -93.2285,B 8.834,C 0.3999,E1 8.828,E2 184.7873} C_DIS
LIN {X -17.1263,Y -138.4235,Z 171,A -95.0875,B 8.8338,C 0.4043,E1 8.8228,E2 186.6783} C_DIS
LIN {X -20.3335,Y -137.9888,Z 171,A -96.2365,B 8.834,C 0.4004,E1 8.8196,E2 187.8044} C_DIS
LIN {X -26.9703,Y -136.8474,Z 171,A -98.8921,B 8.8341,C 0.3972,E1 8.8124,E2 190.4466} C_DIS
LIN {X -35.2843,Y -134.942,Z 171,A -102.5851,B 8.8341,C 0.3989,E1 8.8023,E2 194.1649} C_DIS
LIN {X -39.2423,Y -133.8431,Z 171,A -104.1328,B 8.8342,C 0.3951,E1 8.7982,E2 195.6948} C_DIS
LIN {X -42.6564,Y -132.7946,Z 171,A -105.6208,B 8.8342,C 0.3944,E1 8.7942,E2 197.1858} C_DIS
LIN {X -46.1747,Y -131.6134,Z 171,A -107.0952,B 8.8343,C 0.3922,E1 8.7903,E2 198.654} C_DIS
LIN {X -48.8574,Y -130.6402,Z 171,A -108.3526,B 8.8343,C 0.3927,E1 8.787,E2 199.9224} C_DIS
LIN {X -52.3967,Y -129.2616,Z 171,A -109.8635,B 8.8344,C 0.3903,E1 8.7831,E2 201.4272} C_DIS
LIN {X -55.5058,Y -127.9571,Z 171,A -111.3553,B 8.8344,C 0.3909,E1 8.7792,E2 202.9328} C_DIS
LIN {X -58.7761,Y -126.4884,Z 171,A -112.7248,B 8.8345,C 0.3873,E1 8.7758,E2 204.2891} C_DIS
LIN {X -62.9527,Y -124.4627,Z 171,A -115.4497,B 8.834,C 0.4,E1 8.7687,E2 207.1187} C_DIS
LIN {X -68.2709,Y -121.6287,Z 171,A -116.88,B 8.835,C 0.3778,E1 8.7655,E2 208.415} C_DIS
LIN {X -72.323,Y -119.2638,Z 171,A -119.1833,B 8.8348,C 0.382,E1 8.7599,E2 210.7668} C_DIS
LIN {X -76.0466,Y -116.9246,Z 171,A -120.9712,B 8.8349,C 0.3791,E1 8.7557,E2 212.5521} C_DIS
LIN {X -79.5709,Y -114.5553,Z 171,A -123.1281,B 8.8347,C 0.3838,E1 8.7506,E2 214.7617} C_DIS
LIN {X -82.9251,Y -112.1517,Z 171,A -124.6415,B 8.835,C 0.3778,E1 8.7472,E2 216.2515} C_DIS
LIN {X -86.5783,Y -109.3562,Z 171,A -126.4425,B 8.8352,C 0.373,E1 8.7433,E2 218.0407} C_DIS
LIN {X -90.1803,Y -106.4049,Z 171,A -128.3571,B 8.8352,C 0.3696,E1 8.7392,E2 219.9551} C_DIS
LIN {X -93.6783,Y -103.3383,Z 171,A -130.2642,B 8.8354,C 0.366,E1 8.7352,E2 221.8613} C_DIS
LIN {X -96.9446,Y -100.2806,Z 171,A -132.2893,B 8.8354,C 0.3658,E1 8.7311,E2 223.9097} C_DIS
LIN {X -100.2055,Y -97.0222,Z 171,A -134.1172,B 8.8357,C 0.3609,E1 8.7275,E2 225.7286} C_DIS
LIN {X -105.3228,Y -91.4421,Z 171,A -136.9472,B 8.8361,C 0.3495,E1 8.7223,E2 228.5216} C_DIS
LIN {X -107.296,Y -89.1181,Z 171,A -138.4682,B 8.8361,C 0.3515,E1 8.7195,E2 230.0765} C_DIS
LIN {X -110.048,Y -85.697,Z 171,A -140.3247,B 8.8361,C 0.3484,E1 8.7162,E2 231.939} C_DIS
Enddeposition()
END
